LIN {X 0,Y 171.807,Z 301.135,A -85,B 0,C 180,E1 -23753.467,E2 -23753.467} C_VEL
LIN {X 0,Y 170.77,Z 299.112,A -85,B 0,C 180,E1 -23754.539,E2 -23754.539} C_VEL
LIN {X 0,Y 168.461,Z 295.33,A -85,B 0,C 180,E1 -23756.862,E2 -23756.862} C_VEL
LIN {X 0,Y 167.597,Z 293.95,A -85,B 0,C 180,E1 -23757.747,E2 -23757.747} C_VEL
LIN {X 0,Y 164.577,Z 289.423,A -85,B 0,C 180,E1 -23761.147,E2 -23761.147} C_VEL
LIN {X 0,Y 164.373,Z 288.892,A -85,B 0,C 180,E1 -23761.531,E2 -23761.531} C_VEL
LIN {X 0,Y 163.764,Z 286.973,A -85,B 0,C 180,E1 -23767.397,E2 -23767.397} C_VEL
LIN {X 0,Y 163.542,Z 286.029,A -85,B 0,C 180,E1 -23772.408,E2 -23772.408} C_VEL
LIN {X 0,Y 163.433,Z 285.855,A -85,B 0,C 180,E1 -23777.518,E2 -23777.518} C_VEL
LIN {X 0,Y 163.729,Z 286.439,A -85,B 0,C 180,E1 -23782.726,E2 -23782.726} C_VEL
LIN {X 0,Y 164.407,Z 287.979,A -85,B 0,C 180,E1 -23788.049,E2 -23788.049} C_VEL
LIN {X 0,Y 165.059,Z 289.593,A -85,B 0,C 180,E1 -23791.617,E2 -23791.617} C_VEL
LIN {X 0,Y 166.662,Z 293.516,A -85,B 0,C 180,E1 -23797.542,E2 -23797.542} C_VEL
LIN {X 0,Y 171.614,Z 300.55,A -85,B 0,C 180,E1 -23801.978,E2 -23801.978} C_VEL
LIN {X 0,Y 174.691,Z 306.548,A -85,B 0,C 180,E1 -23804.603,E2 -23804.603} C_VEL
LIN {X 0,Y 176.775,Z 311.643,A -85,B 0,C 180,E1 -23806.516,E2 -23806.516} C_VEL
LIN {X 0,Y 178.262,Z 321.519,A -85,B 0,C 180,E1 -23809.162,E2 -23809.162} C_VEL
LIN {X 0,Y 178.652,Z 330.917,A -85,B 0,C 180,E1 -23811.605,E2 -23811.605} C_VEL
LIN {X 0,Y 178.13,Z 336.639,A -85,B 0,C 180,E1 -23813.07,E2 -23813.07} C_VEL
LIN {X 0,Y 175.624,Z 345.707,A -85,B 0,C 180,E1 -23815.233,E2 -23815.233} C_VEL
LIN {X 0,Y 173.203,Z 353.233,A -85,B 0,C 180,E1 -23817.477,E2 -23817.477} C_VEL
LIN {X 0,Y 169.307,Z 361.018,A -85,B 0,C 180,E1 -23820.124,E2 -23820.124} C_VEL
LIN {X 0,Y 166.418,Z 366.182,A -85,B 0,C 180,E1 -23822.32,E2 -23822.32} C_VEL
LIN {X 0,Y 163.949,Z 370.527,A -85,B 0,C 180,E1 -23824.617,E2 -23824.617} C_VEL
LIN {X 0,Y 160.848,Z 375.707,A -85,B 0,C 180,E1 -23828.199,E2 -23828.199} C_VEL
LIN {X 0,Y 158.228,Z 379.6,A -85,B 0,C 180,E1 -23831.886,E2 -23831.886} C_VEL
LIN {X 0,Y 156.906,Z 381.458,A -85,B 0,C 180,E1 -23834.411,E2 -23834.411} C_VEL
LIN {X 0,Y 156.007,Z 382.844,A -85,B 0,C 180,E1 -23836.983,E2 -23836.983} C_VEL
LIN {X 0,Y 155.411,Z 383.78,A -85,B 0,C 180,E1 -23839.579,E2 -23839.579} C_VEL
LIN {X 0,Y 155.045,Z 384.215,A -85,B 0,C 180,E1 -23842.185,E2 -23842.185} C_VEL
LIN {X 0,Y 155.037,Z 383.994,A -85,B 0,C 180,E1 -23845.776,E2 -23845.776} C_VEL
LIN {X 0,Y 155.371,Z 382.438,A -85,B 0,C 180,E1 -23850,E2 -23850} C_VEL
LIN {X 0,Y 155.426,Z 380.832,A -85,B 0,C 180,E1 -23852.592,E2 -23852.592} C_VEL
LIN {X 0,Y 155.785,Z 377.198,A -85,B 0,C 180,E1 -23856.476,E2 -23856.476} C_VEL
LIN {X 0,Y 156.411,Z 374.594,A -85,B 0,C 180,E1 -23858.772,E2 -23858.772} C_VEL
LIN {X 0,Y 156.872,Z 377.363,A -85,B 0,C 180,E1 -23862.945,E2 -23862.945} C_VEL
LIN {X 0,Y 158.749,Z 379.707,A -85,B 0,C 180,E1 -23868.054,E2 -23868.054} C_VEL
LIN {X 0,Y 162.293,Z 380.986,A -85,B 0,C 180,E1 -23872.939,E2 -23872.939} C_VEL
LIN {X 0,Y 167.198,Z 381.193,A -85,B 0,C 180,E1 -23877.541,E2 -23877.541} C_VEL
LIN {X 0,Y 170.684,Z 380.806,A -85,B 0,C 180,E1 -23880.126,E2 -23880.126} C_VEL
LIN {X 0,Y 172.842,Z 380.336,A -85,B 0,C 180,E1 -23881.957,E2 -23881.957} C_VEL
LIN {X 0,Y 177.848,Z 378.2,A -85,B 0,C 180,E1 -23887.502,E2 -23887.502} C_VEL
LIN {X 0,Y 180.635,Z 377.227,A -85,B 0,C 180,E1 -23889.123,E2 -23889.123} C_VEL
LIN {X 0,Y 181.821,Z 376.834,A -85,B 0,C 180,E1 -23889.601,E2 -23889.601} C_VEL
LIN {X 0,Y 189.036,Z 374.503,A -85,B 0,C 180,E1 -23892.007,E2 -23892.007} C_VEL
LIN {X 0,Y 193.684,Z 372.683,A -85,B 0,C 180,E1 -23893.586,E2 -23893.586} C_VEL
LIN {X 0,Y 196.724,Z 371.102,A -85,B 0,C 180,E1 -23895.603,E2 -23895.603} C_VEL
LIN {X 0,Y 197.955,Z 370.173,A -85,B 0,C 180,E1 -23897.58,E2 -23897.58} C_VEL
LIN {X 0,Y 198.038,Z 370.015,A -85,B 0,C 180,E1 -23898.182,E2 -23898.182} C_VEL
LIN {X 0,Y 197.073,Z 370.011,A -85,B 0,C 180,E1 -23900.065,E2 -23900.065} C_VEL
LIN {X 0,Y 192.395,Z 371.253,A -85,B 0,C 180,E1 -23901.611,E2 -23901.611} C_VEL
LIN {X 0,Y 182.935,Z 373.108,A -85,B 0,C 180,E1 -23904.812,E2 -23904.812} C_VEL
LIN {X 0,Y 174.413,Z 373.822,A -85,B 0,C 180,E1 -23908.41,E2 -23908.41} C_VEL
LIN {X 0,Y 166.91,Z 373.402,A -85,B 0,C 180,E1 -23912.408,E2 -23912.408} C_VEL
LIN {X 0,Y 160.609,Z 371.833,A -85,B 0,C 180,E1 -23916.807,E2 -23916.807} C_VEL
LIN {X 0,Y 155.459,Z 369.106,A -85,B 0,C 180,E1 -23921.551,E2 -23921.551} C_VEL
LIN {X 0,Y 152.113,Z 365.227,A -85,B 0,C 180,E1 -23926.644,E2 -23926.644} C_VEL
LIN {X 0,Y 150.015,Z 360.025,A -85,B 0,C 180,E1 -23931.921,E2 -23931.921} C_VEL
LIN {X 0,Y 148.825,Z 353.277,A -85,B 0,C 180,E1 -23937.294,E2 -23937.294} C_VEL
LIN {X 0,Y 148.718,Z 345.944,A -85,B 0,C 180,E1 -23942.031,E2 -23942.031} C_VEL
LIN {X 0,Y 149.01,Z 337.459,A -85,B 0,C 180,E1 -23946.444,E2 -23946.444} C_VEL
LIN {X 0,Y 149.593,Z 328.841,A -85,B 0,C 180,E1 -23950.147,E2 -23950.147} C_VEL
LIN {X 0,Y 150.594,Z 317.422,A -85,B 0,C 180,E1 -23954.183,E2 -23954.183} C_VEL
LIN {X 0,Y 151.665,Z 306.976,A -85,B 0,C 180,E1 -23957.183,E2 -23957.183} C_VEL
LIN {X 0,Y 153,Z 294.302,A -85,B 0,C 180,E1 -23960.152,E2 -23960.152} C_VEL
LIN {X 0,Y 150.87,Z 281.95,A -85,B 0,C 180,E1 -23962.402,E2 -23962.402} C_VEL
LIN {X 0,Y 149.044,Z 269.969,A -85,B 0,C 180,E1 -23964.182,E2 -23964.182} C_VEL
LIN {X 0,Y 149.609,Z 269.848,A -85,B 0,C 180,E1 -23972.267,E2 -23972.267} C_VEL
LIN {X 0,Y 149.987,Z 269.803,A -85,B 0,C 180,E1 -23977.528,E2 -23977.528} C_VEL
LIN {X 0,Y 150.097,Z 269.785,A -85,B 0,C 180,E1 -23981.481,E2 -23981.481} C_VEL
LIN {X 0,Y 150.128,Z 269.785,A -85,B 0,C 180,E1 -23985.395,E2 -23985.395} C_VEL
LIN {X 0,Y 150.14,Z 269.784,A -85,B 0,C 180,E1 -23989.054,E2 -23989.054} C_VEL
LIN {X 0,Y 150.178,Z 269.777,A -85,B 0,C 180,E1 -23992.71,E2 -23992.71} C_VEL
LIN {X 0,Y 150.207,Z 269.774,A -85,B 0,C 180,E1 -23997.374,E2 -23997.374} C_VEL
LIN {X 0,Y 150.241,Z 269.771,A -85,B 0,C 180,E1 -24002.722,E2 -24002.722} C_VEL
LIN {X 0,Y 150.352,Z 269.756,A -85,B 0,C 180,E1 -24009.209,E2 -24009.209} C_VEL
LIN {X 0,Y 150.364,Z 269.748,A -85,B 0,C 180,E1 -24013.713,E2 -24013.713} C_VEL
LIN {X 0,Y 150.613,Z 269.726,A -85,B 0,C 180,E1 -24019.242,E2 -24019.242} C_VEL
LIN {X 0,Y 150.701,Z 269.791,A -85,B 0,C 180,E1 -24022.968,E2 -24022.968} C_VEL
LIN {X 0,Y 152.144,Z 275.605,A -85,B 0,C 180,E1 -24028.676,E2 -24028.676} C_VEL
LIN {X 0,Y 152.345,Z 278.494,A -85,B 0,C 180,E1 -24031.321,E2 -24031.321} C_VEL
LIN {X 0,Y 151.838,Z 283.129,A -85,B 0,C 180,E1 -24035.311,E2 -24035.311} C_VEL
LIN {X 0,Y 151.536,Z 285.299,A -85,B 0,C 180,E1 -24037.16,E2 -24037.16} C_VEL
LIN {X 0,Y 153.606,Z 296.207,A -85,B 0,C 180,E1 -24038.551,E2 -24038.551} C_VEL
LIN {X 0,Y 154.832,Z 304.081,A -85,B 0,C 180,E1 -24039.8,E2 -24039.8} C_VEL
LIN {X 0,Y 155.768,Z 312.475,A -85,B 0,C 180,E1 -24041.384,E2 -24041.384} C_VEL
LIN {X 0,Y 156.371,Z 319.655,A -85,B 0,C 180,E1 -24042.986,E2 -24042.986} C_VEL
LIN {X 0,Y 155.521,Z 325.645,A -85,B 0,C 180,E1 -24044.391,E2 -24044.391} C_VEL
LIN {X 0,Y 153.97,Z 333.329,A -85,B 0,C 180,E1 -24046.552,E2 -24046.552} C_VEL
LIN {X 0,Y 152.622,Z 339.884,A -85,B 0,C 180,E1 -24048.804,E2 -24048.804} C_VEL
LIN {X 0,Y 151.181,Z 346.539,A -85,B 0,C 180,E1 -24051.603,E2 -24051.603} C_VEL
LIN {X 0,Y 149.791,Z 352.955,A -85,B 0,C 180,E1 -24054.978,E2 -24054.978} C_VEL
LIN {X 0,Y 148.818,Z 357.754,A -85,B 0,C 180,E1 -24058.18,E2 -24058.18} C_VEL
LIN {X 0,Y 148.1,Z 361.611,A -85,B 0,C 180,E1 -24061.466,E2 -24061.466} C_VEL
LIN {X 0,Y 147.702,Z 365.391,A -85,B 0,C 180,E1 -24066.011,E2 -24066.011} C_VEL
LIN {X 0,Y 147.758,Z 366.729,A -85,B 0,C 180,E1 -24068.194,E2 -24068.194} C_VEL
LIN {X 0,Y 148.185,Z 368.093,A -85,B 0,C 180,E1 -24071.604,E2 -24071.604} C_VEL
LIN {X 0,Y 149.05,Z 368.678,A -85,B 0,C 180,E1 -24075.014,E2 -24075.014} C_VEL
LIN {X 0,Y 150.744,Z 368.281,A -85,B 0,C 180,E1 -24079.253,E2 -24079.253} C_VEL
LIN {X 0,Y 153.066,Z 366.635,A -85,B 0,C 180,E1 -24083.352,E2 -24083.352} C_VEL
LIN {X 0,Y 154.299,Z 365.627,A -85,B 0,C 180,E1 -24085.071,E2 -24085.071} C_VEL
LIN {X 0,Y 156.967,Z 362.887,A -85,B 0,C 180,E1 -24088.288,E2 -24088.288} C_VEL
LIN {X 0,Y 160.032,Z 359.11,A -85,B 0,C 180,E1 -24091.441,E2 -24091.441} C_VEL
LIN {X 0,Y 163.779,Z 353.917,A -85,B 0,C 180,E1 -24094.588,E2 -24094.588} C_VEL
LIN {X 0,Y 167.587,Z 347.987,A -85,B 0,C 180,E1 -24097.309,E2 -24097.309} C_VEL
LIN {X 0,Y 170.971,Z 341.922,A -85,B 0,C 180,E1 -24099.504,E2 -24099.504} C_VEL
LIN {X 0,Y 172.124,Z 339.009,A -85,B 0,C 180,E1 -24100.552,E2 -24100.552} C_VEL
LIN {X 0,Y 173.216,Z 331.259,A -85,B 0,C 180,E1 -24103.5,E2 -24103.5} C_VEL
LIN {X 0,Y 173.37,Z 324.684,A -85,B 0,C 180,E1 -24105.923,E2 -24105.923} C_VEL
LIN {X 0,Y 172.775,Z 318.629,A -85,B 0,C 180,E1 -24108.265,E2 -24108.265} C_VEL
LIN {X 0,Y 170.637,Z 312.341,A -85,B 0,C 180,E1 -24111.296,E2 -24111.296} C_VEL
LIN {X 0,Y 167.582,Z 305.138,A -85,B 0,C 180,E1 -24115.188,E2 -24115.188} C_VEL
LIN {X 0,Y 165.383,Z 301.117,A -85,B 0,C 180,E1 -24117.793,E2 -24117.793} C_VEL
LIN {X 0,Y 161.882,Z 295.216,A -85,B 0,C 180,E1 -24122.488,E2 -24122.488} C_VEL
LIN {X 0,Y 158.701,Z 291.959,A -85,B 0,C 180,E1 -24127.474,E2 -24127.474} C_VEL
LIN {X 0,Y 157.556,Z 290.073,A -85,B 0,C 180,E1 -24130.278,E2 -24130.278} C_VEL
LIN {X 0,Y 157.464,Z 289.678,A -85,B 0,C 180,E1 -24135.533,E2 -24135.533} C_VEL
LIN {X 0,Y 157.647,Z 290.116,A -85,B 0,C 180,E1 -24140.894,E2 -24140.894} C_VEL
LIN {X 0,Y 158.302,Z 291.389,A -85,B 0,C 180,E1 -24146.357,E2 -24146.357} C_VEL
LIN {X 0,Y 158.745,Z 292.495,A -85,B 0,C 180,E1 -24148.928,E2 -24148.928} C_VEL
LIN {X 0,Y 164.433,Z 300.122,A -85,B 0,C 180,E1 -24156.908,E2 -24156.908} C_VEL
LIN {X 0,Y 168.556,Z 306.487,A -85,B 0,C 180,E1 -24161.126,E2 -24161.126} C_VEL
LIN {X 0,Y 170.828,Z 311.443,A -85,B 0,C 180,E1 -24163.478,E2 -24163.478} C_VEL
LIN {X 0,Y 172.505,Z 316.408,A -85,B 0,C 180,E1 -24165.478,E2 -24165.478} C_VEL
LIN {X 0,Y 173.332,Z 325.826,A -85,B 0,C 180,E1 -24168.2,E2 -24168.2} C_VEL
LIN {X 0,Y 173.204,Z 333.712,A -85,B 0,C 180,E1 -24170.439,E2 -24170.439} C_VEL
LIN {X 0,Y 172.921,Z 337.214,A -85,B 0,C 180,E1 -24171.413,E2 -24171.413} C_VEL
LIN {X 0,Y 169.917,Z 346.903,A -85,B 0,C 180,E1 -24173.886,E2 -24173.886} C_VEL
LIN {X 0,Y 167.304,Z 354.116,A -85,B 0,C 180,E1 -24176.179,E2 -24176.179} C_VEL
LIN {X 0,Y 164.023,Z 360.283,A -85,B 0,C 180,E1 -24178.34,E2 -24178.34} C_VEL
LIN {X 0,Y 160.181,Z 366.633,A -85,B 0,C 180,E1 -24181.143,E2 -24181.143} C_VEL
LIN {X 0,Y 157.566,Z 370.826,A -85,B 0,C 180,E1 -24183.511,E2 -24183.511} C_VEL
LIN {X 0,Y 154.271,Z 375.865,A -85,B 0,C 180,E1 -24187.218,E2 -24187.218} C_VEL
LIN {X 0,Y 151.491,Z 379.605,A -85,B 0,C 180,E1 -24191.05,E2 -24191.05} C_VEL
LIN {X 0,Y 150.042,Z 381.346,A -85,B 0,C 180,E1 -24193.678,E2 -24193.678} C_VEL
LIN {X 0,Y 149.06,Z 382.615,A -85,B 0,C 180,E1 -24196.365,E2 -24196.365} C_VEL
LIN {X 0,Y 148.388,Z 383.441,A -85,B 0,C 180,E1 -24199.08,E2 -24199.08} C_VEL
LIN {X 0,Y 147.991,Z 383.82,A -85,B 0,C 180,E1 -24201.81,E2 -24201.81} C_VEL
LIN {X 0,Y 147.977,Z 383.385,A -85,B 0,C 180,E1 -24205.844,E2 -24205.844} C_VEL
LIN {X 0,Y 148.306,Z 381.789,A -85,B 0,C 180,E1 -24210,E2 -24210} C_VEL
LIN {X 0,Y 148.407,Z 378.972,A -85,B 0,C 180,E1 -24214.074,E2 -24214.074} C_VEL
LIN {X 0,Y 149.086,Z 374.871,A -85,B 0,C 180,E1 -24218.131,E2 -24218.131} C_VEL
LIN {X 0,Y 149.621,Z 373.086,A -85,B 0,C 180,E1 -24219.634,E2 -24219.634} C_VEL
LIN {X 0,Y 150.119,Z 375.704,A -85,B 0,C 180,E1 -24223.538,E2 -24223.538} C_VEL
LIN {X 0,Y 152.121,Z 378.357,A -85,B 0,C 180,E1 -24228.869,E2 -24228.869} C_VEL
LIN {X 0,Y 155.822,Z 379.961,A -85,B 0,C 180,E1 -24233.95,E2 -24233.95} C_VEL
LIN {X 0,Y 160.959,Z 380.526,A -85,B 0,C 180,E1 -24238.705,E2 -24238.705} C_VEL
LIN {X 0,Y 167.382,Z 380.073,A -85,B 0,C 180,E1 -24243.083,E2 -24243.083} C_VEL
LIN {X 0,Y 175.194,Z 378.621,A -85,B 0,C 180,E1 -24246.995,E2 -24246.995} C_VEL
LIN {X 0,Y 181.821,Z 376.834,A -85,B 0,C 180,E1 -24249.601,E2 -24249.601} C_VEL
LIN {X 0,Y 193.185,Z 372.928,A -85,B 0,C 180,E1 -24253.315,E2 -24253.315} C_VEL
LIN {X 0,Y 194.417,Z 372.367,A -85,B 0,C 180,E1 -24253.96,E2 -24253.96} C_VEL
LIN {X 0,Y 194.868,Z 371.948,A -85,B 0,C 180,E1 -24254.912,E2 -24254.912} C_VEL
LIN {X 0,Y 194.1,Z 371.779,A -85,B 0,C 180,E1 -24256.298,E2 -24256.298} C_VEL
LIN {X 0,Y 191.77,Z 372.044,A -85,B 0,C 180,E1 -24257.97,E2 -24257.97} C_VEL
LIN {X 0,Y 188.64,Z 372.559,A -85,B 0,C 180,E1 -24259.544,E2 -24259.544} C_VEL
LIN {X 0,Y 186.99,Z 372.866,A -85,B 0,C 180,E1 -24260.287,E2 -24260.287} C_VEL
LIN {X 0,Y 177.233,Z 374.236,A -85,B 0,C 180,E1 -24263.501,E2 -24263.501} C_VEL
LIN {X 0,Y 168.427,Z 374.487,A -85,B 0,C 180,E1 -24267.149,E2 -24267.149} C_VEL
LIN {X 0,Y 160.661,Z 373.62,A -85,B 0,C 180,E1 -24271.237,E2 -24271.237} C_VEL
LIN {X 0,Y 154.111,Z 371.633,A -85,B 0,C 180,E1 -24275.768,E2 -24275.768} C_VEL
LIN {X 0,Y 148.775,Z 368.506,A -85,B 0,C 180,E1 -24280.69,E2 -24280.69} C_VEL
LIN {X 0,Y 145.282,Z 364.241,A -85,B 0,C 180,E1 -24286.003,E2 -24286.003} C_VEL
LIN {X 0,Y 143.116,Z 358.694,A -85,B 0,C 180,E1 -24291.529,E2 -24291.529} C_VEL
LIN {X 0,Y 141.911,Z 351.525,A -85,B 0,C 180,E1 -24297.162,E2 -24297.162} C_VEL
LIN {X 0,Y 141.817,Z 344.989,A -85,B 0,C 180,E1 -24301.42,E2 -24301.42} C_VEL
LIN {X 0,Y 142.044,Z 337.093,A -85,B 0,C 180,E1 -24305.679,E2 -24305.679} C_VEL
LIN {X 0,Y 142.578,Z 328.22,A -85,B 0,C 180,E1 -24309.647,E2 -24309.647} C_VEL
LIN {X 0,Y 143.562,Z 316.905,A -85,B 0,C 180,E1 -24313.807,E2 -24313.807} C_VEL
LIN {X 0,Y 144.742,Z 305.089,A -85,B 0,C 180,E1 -24317.302,E2 -24317.302} C_VEL
LIN {X 0,Y 145.846,Z 293.735,A -85,B 0,C 180,E1 -24320.046,E2 -24320.046} C_VEL
LIN {X 0,Y 143.451,Z 280.113,A -85,B 0,C 180,E1 -24322.57,E2 -24322.57} C_VEL
LIN {X 0,Y 142.01,Z 270.797,A -85,B 0,C 180,E1 -24324.001,E2 -24324.001} C_VEL
LIN {X 0,Y 142.251,Z 270.764,A -85,B 0,C 180,E1 -24329.608,E2 -24329.608} C_VEL
LIN {X 0,Y 142.62,Z 270.717,A -85,B 0,C 180,E1 -24333.098,E2 -24333.098} C_VEL
LIN {X 0,Y 142.923,Z 270.682,A -85,B 0,C 180,E1 -24338.114,E2 -24338.114} C_VEL
LIN {X 0,Y 143.025,Z 270.672,A -85,B 0,C 180,E1 -24343.468,E2 -24343.468} C_VEL
LIN {X 0,Y 143.04,Z 270.664,A -85,B 0,C 180,E1 -24347.477,E2 -24347.477} C_VEL
LIN {X 0,Y 143.074,Z 270.664,A -85,B 0,C 180,E1 -24351.809,E2 -24351.809} C_VEL
LIN {X 0,Y 143.175,Z 270.65,A -85,B 0,C 180,E1 -24357.319,E2 -24357.319} C_VEL
LIN {X 0,Y 143.185,Z 270.65,A -85,B 0,C 180,E1 -24362.069,E2 -24362.069} C_VEL
LIN {X 0,Y 143.278,Z 270.638,A -85,B 0,C 180,E1 -24368.747,E2 -24368.747} C_VEL
LIN {X 0,Y 143.304,Z 270.624,A -85,B 0,C 180,E1 -24372.886,E2 -24372.886} C_VEL
LIN {X 0,Y 143.539,Z 270.604,A -85,B 0,C 180,E1 -24378.705,E2 -24378.705} C_VEL
LIN {X 0,Y 143.679,Z 270.713,A -85,B 0,C 180,E1 -24381.915,E2 -24381.915} C_VEL
LIN {X 0,Y 145.241,Z 277.269,A -85,B 0,C 180,E1 -24388.613,E2 -24388.613} C_VEL
LIN {X 0,Y 145.388,Z 280.234,A -85,B 0,C 180,E1 -24391.385,E2 -24391.385} C_VEL
LIN {X 0,Y 144.683,Z 285.645,A -85,B 0,C 180,E1 -24396.187,E2 -24396.187} C_VEL
LIN {X 0,Y 146.749,Z 296.639,A -85,B 0,C 180,E1 -24397.654,E2 -24397.654} C_VEL
LIN {X 0,Y 148.158,Z 305.851,A -85,B 0,C 180,E1 -24399.212,E2 -24399.212} C_VEL
LIN {X 0,Y 149.139,Z 315.612,A -85,B 0,C 180,E1 -24401.208,E2 -24401.208} C_VEL
LIN {X 0,Y 149.475,Z 321.134,A -85,B 0,C 180,E1 -24402.559,E2 -24402.559} C_VEL
LIN {X 0,Y 147.825,Z 329.804,A -85,B 0,C 180,E1 -24404.805,E2 -24404.805} C_VEL
LIN {X 0,Y 146.118,Z 338.047,A -85,B 0,C 180,E1 -24407.494,E2 -24407.494} C_VEL
LIN {X 0,Y 144.469,Z 345.364,A -85,B 0,C 180,E1 -24410.546,E2 -24410.546} C_VEL
LIN {X 0,Y 143.039,Z 351.765,A -85,B 0,C 180,E1 -24413.913,E2 -24413.913} C_VEL
LIN {X 0,Y 142.009,Z 356.514,A -85,B 0,C 180,E1 -24417.022,E2 -24417.022} C_VEL
LIN {X 0,Y 141.082,Z 361.178,A -85,B 0,C 180,E1 -24420.914,E2 -24420.914} C_VEL
LIN {X 0,Y 140.636,Z 364.881,A -85,B 0,C 180,E1 -24425.078,E2 -24425.078} C_VEL
LIN {X 0,Y 140.899,Z 367.803,A -85,B 0,C 180,E1 -24430.423,E2 -24430.423} C_VEL
LIN {X 0,Y 141.62,Z 368.809,A -85,B 0,C 180,E1 -24434.008,E2 -24434.008} C_VEL
LIN {X 0,Y 142.813,Z 369.031,A -85,B 0,C 180,E1 -24437.575,E2 -24437.575} C_VEL
LIN {X 0,Y 144.494,Z 368.463,A -85,B 0,C 180,E1 -24441.098,E2 -24441.098} C_VEL
LIN {X 0,Y 147.951,Z 366.08,A -85,B 0,C 180,E1 -24446.353,E2 -24446.353} C_VEL
LIN {X 0,Y 151.119,Z 362.993,A -85,B 0,C 180,E1 -24450.041,E2 -24450.041} C_VEL
LIN {X 0,Y 154.779,Z 358.723,A -85,B 0,C 180,E1 -24453.53,E2 -24453.53} C_VEL
LIN {X 0,Y 158.579,Z 353.787,A -85,B 0,C 180,E1 -24456.492,E2 -24456.492} C_VEL
LIN {X 0,Y 162.895,Z 347.427,A -85,B 0,C 180,E1 -24459.387,E2 -24459.387} C_VEL
LIN {X 0,Y 165.436,Z 343.103,A -85,B 0,C 180,E1 -24460.957,E2 -24460.957} C_VEL
LIN {X 0,Y 166.599,Z 339.938,A -85,B 0,C 180,E1 -24462.25,E2 -24462.25} C_VEL
LIN {X 0,Y 167.825,Z 332.05,A -85,B 0,C 180,E1 -24465.447,E2 -24465.447} C_VEL
LIN {X 0,Y 168.122,Z 325.849,A -85,B 0,C 180,E1 -24467.935,E2 -24467.935} C_VEL
LIN {X 0,Y 167.604,Z 321.749,A -85,B 0,C 180,E1 -24469.772,E2 -24469.772} C_VEL
LIN {X 0,Y 165.583,Z 315.244,A -85,B 0,C 180,E1 -24473.297,E2 -24473.297} C_VEL
LIN {X 0,Y 163.637,Z 310.341,A -85,B 0,C 180,E1 -24476.306,E2 -24476.306} C_VEL
LIN {X 0,Y 161.264,Z 305.387,A -85,B 0,C 180,E1 -24480,E2 -24480} C_VEL
LIN {X 0,Y 159.406,Z 301.654,A -85,B 0,C 180,E1 -24483.159,E2 -24483.159} C_VEL
LIN {X 0,Y 156.829,Z 298.625,A -85,B 0,C 180,E1 -24488.043,E2 -24488.043} C_VEL
LIN {X 0,Y 155.867,Z 296.907,A -85,B 0,C 180,E1 -24490.785,E2 -24490.785} C_VEL
LIN {X 0,Y 154.56,Z 296.202,A -85,B 0,C 180,E1 -24497.275,E2 -24497.275} C_VEL
LIN {X 0,Y 155.145,Z 297.123,A -85,B 0,C 180,E1 -24503.351,E2 -24503.351} C_VEL
LIN {X 0,Y 156.989,Z 299.239,A -85,B 0,C 180,E1 -24508.416,E2 -24508.416} C_VEL
LIN {X 0,Y 161.888,Z 306.537,A -85,B 0,C 180,E1 -24516.263,E2 -24516.263} C_VEL
LIN {X 0,Y 164.993,Z 311.624,A -85,B 0,C 180,E1 -24519.939,E2 -24519.939} C_VEL
LIN {X 0,Y 167.257,Z 317.894,A -85,B 0,C 180,E1 -24523.064,E2 -24523.064} C_VEL
LIN {X 0,Y 168.166,Z 321.202,A -85,B 0,C 180,E1 -24524.43,E2 -24524.43} C_VEL
LIN {X 0,Y 168.25,Z 331.7,A -85,B 0,C 180,E1 -24527.716,E2 -24527.716} C_VEL
LIN {X 0,Y 167.536,Z 338.916,A -85,B 0,C 180,E1 -24529.927,E2 -24529.927} C_VEL
LIN {X 0,Y 165.062,Z 346.196,A -85,B 0,C 180,E1 -24531.875,E2 -24531.875} C_VEL
LIN {X 0,Y 162.266,Z 353.413,A -85,B 0,C 180,E1 -24534.218,E2 -24534.218} C_VEL
LIN {X 0,Y 158.925,Z 359.605,A -85,B 0,C 180,E1 -24536.442,E2 -24536.442} C_VEL
LIN {X 0,Y 154.792,Z 365.997,A -85,B 0,C 180,E1 -24539.284,E2 -24539.284} C_VEL
LIN {X 0,Y 152.49,Z 369.354,A -85,B 0,C 180,E1 -24541.125,E2 -24541.125} C_VEL
LIN {X 0,Y 148.786,Z 374.513,A -85,B 0,C 180,E1 -24544.842,E2 -24544.842} C_VEL
LIN {X 0,Y 145.672,Z 378.469,A -85,B 0,C 180,E1 -24548.787,E2 -24548.787} C_VEL
LIN {X 0,Y 143.209,Z 381.249,A -85,B 0,C 180,E1 -24552.876,E2 -24552.876} C_VEL
LIN {X 0,Y 142.141,Z 382.398,A -85,B 0,C 180,E1 -24555.687,E2 -24555.687} C_VEL
LIN {X 0,Y 141.39,Z 383.105,A -85,B 0,C 180,E1 -24558.532,E2 -24558.532} C_VEL
LIN {X 0,Y 140.959,Z 383.378,A -85,B 0,C 180,E1 -24561.398,E2 -24561.398} C_VEL
LIN {X 0,Y 140.92,Z 382.758,A -85,B 0,C 180,E1 -24565.905,E2 -24565.905} C_VEL
LIN {X 0,Y 141.242,Z 381.13,A -85,B 0,C 180,E1 -24570,E2 -24570} C_VEL
LIN {X 0,Y 141.37,Z 378.201,A -85,B 0,C 180,E1 -24574.277,E2 -24574.277} C_VEL
LIN {X 0,Y 142.133,Z 373.909,A -85,B 0,C 180,E1 -24578.531,E2 -24578.531} C_VEL
LIN {X 0,Y 142.931,Z 371.413,A -85,B 0,C 180,E1 -24580.537,E2 -24580.537} C_VEL
LIN {X 0,Y 144.27,Z 375.536,A -85,B 0,C 180,E1 -24586.995,E2 -24586.995} C_VEL
LIN {X 0,Y 147.273,Z 377.973,A -85,B 0,C 180,E1 -24592.444,E2 -24592.444} C_VEL
LIN {X 0,Y 151.905,Z 379.387,A -85,B 0,C 180,E1 -24597.559,E2 -24597.559} C_VEL
LIN {X 0,Y 157.935,Z 379.801,A -85,B 0,C 180,E1 -24602.276,E2 -24602.276} C_VEL
LIN {X 0,Y 165.338,Z 379.252,A -85,B 0,C 180,E1 -24606.52,E2 -24606.52} C_VEL
LIN {X 0,Y 174.109,Z 377.723,A -85,B 0,C 180,E1 -24610.23,E2 -24610.23} C_VEL
LIN {X 0,Y 183.85,Z 375.192,A -85,B 0,C 180,E1 -24613.479,E2 -24613.479} C_VEL
LIN {X 0,Y 188.392,Z 373.65,A -85,B 0,C 180,E1 -24615.138,E2 -24615.138} C_VEL
LIN {X 0,Y 190.893,Z 372.403,A -85,B 0,C 180,E1 -24617.42,E2 -24617.42} C_VEL
LIN {X 0,Y 191.006,Z 372.128,A -85,B 0,C 180,E1 -24618.524,E2 -24618.524} C_VEL
LIN {X 0,Y 188.64,Z 372.559,A -85,B 0,C 180,E1 -24619.544,E2 -24619.544} C_VEL
LIN {X 0,Y 186.325,Z 373.029,A -85,B 0,C 180,E1 -24620.237,E2 -24620.237} C_VEL
LIN {X 0,Y 182.184,Z 373.821,A -85,B 0,C 180,E1 -24620.871,E2 -24620.871} C_VEL
LIN {X 0,Y 173.219,Z 375.04,A -85,B 0,C 180,E1 -24621.899,E2 -24621.899} C_VEL
LIN {X 0,Y 169.993,Z 375.2,A -85,B 0,C 180,E1 -24622.709,E2 -24622.709} C_VEL
LIN {X 0,Y 162.529,Z 374.98,A -85,B 0,C 180,E1 -24625.796,E2 -24625.796} C_VEL
LIN {X 0,Y 154.472,Z 373.673,A -85,B 0,C 180,E1 -24629.969,E2 -24629.969} C_VEL
LIN {X 0,Y 147.683,Z 371.272,A -85,B 0,C 180,E1 -24634.641,E2 -24634.641} C_VEL
LIN {X 0,Y 142.148,Z 367.74,A -85,B 0,C 180,E1 -24639.752,E2 -24639.752} C_VEL
LIN {X 0,Y 138.512,Z 363.094,A -85,B 0,C 180,E1 -24645.304,E2 -24645.304} C_VEL
LIN {X 0,Y 136.241,Z 357.148,A -85,B 0,C 180,E1 -24651.098,E2 -24651.098} C_VEL
LIN {X 0,Y 135.054,Z 349.606,A -85,B 0,C 180,E1 -24657.017,E2 -24657.017} C_VEL
LIN {X 0,Y 134.959,Z 342.701,A -85,B 0,C 180,E1 -24661.492,E2 -24661.492} C_VEL
LIN {X 0,Y 135.202,Z 334.358,A -85,B 0,C 180,E1 -24665.968,E2 -24665.968} C_VEL
LIN {X 0,Y 135.773,Z 324.969,A -85,B 0,C 180,E1 -24670.135,E2 -24670.135} C_VEL
LIN {X 0,Y 136.749,Z 314.063,A -85,B 0,C 180,E1 -24674.13,E2 -24674.13} C_VEL
LIN {X 0,Y 137.987,Z 301.65,A -85,B 0,C 180,E1 -24677.794,E2 -24677.794} C_VEL
LIN {X 0,Y 138.706,Z 293.442,A -85,B 0,C 180,E1 -24679.807,E2 -24679.807} C_VEL
LIN {X 0,Y 136.238,Z 279.723,A -85,B 0,C 180,E1 -24682.454,E2 -24682.454} C_VEL
LIN {X 0,Y 134.981,Z 271.673,A -85,B 0,C 180,E1 -24683.803,E2 -24683.803} C_VEL
LIN {X 0,Y 135.339,Z 271.627,A -85,B 0,C 180,E1 -24691.285,E2 -24691.285} C_VEL
LIN {X 0,Y 135.633,Z 271.583,A -85,B 0,C 180,E1 -24694.749,E2 -24694.749} C_VEL
LIN {X 0,Y 135.922,Z 271.554,A -85,B 0,C 180,E1 -24699.14,E2 -24699.14} C_VEL
LIN {X 0,Y 135.971,Z 271.55,A -85,B 0,C 180,E1 -24703.644,E2 -24703.644} C_VEL
LIN {X 0,Y 135.984,Z 271.543,A -85,B 0,C 180,E1 -24707.787,E2 -24707.787} C_VEL
LIN {X 0,Y 136.023,Z 271.542,A -85,B 0,C 180,E1 -24711.682,E2 -24711.682} C_VEL
LIN {X 0,Y 136.053,Z 271.539,A -85,B 0,C 180,E1 -24715.742,E2 -24715.742} C_VEL
LIN {X 0,Y 136.142,Z 271.527,A -85,B 0,C 180,E1 -24722.315,E2 -24722.315} C_VEL
LIN {X 0,Y 136.244,Z 271.514,A -85,B 0,C 180,E1 -24728.832,E2 -24728.832} C_VEL
LIN {X 0,Y 136.271,Z 271.511,A -85,B 0,C 180,E1 -24735.056,E2 -24735.056} C_VEL
LIN {X 0,Y 136.536,Z 271.541,A -85,B 0,C 180,E1 -24740.658,E2 -24740.658} C_VEL
LIN {X 0,Y 137.529,Z 276.19,A -85,B 0,C 180,E1 -24745.603,E2 -24745.603} C_VEL
LIN {X 0,Y 138.354,Z 278.95,A -85,B 0,C 180,E1 -24748.544,E2 -24748.544} C_VEL
LIN {X 0,Y 138.416,Z 281.946,A -85,B 0,C 180,E1 -24751.454,E2 -24751.454} C_VEL
LIN {X 0,Y 137.878,Z 286.1,A -85,B 0,C 180,E1 -24755.117,E2 -24755.117} C_VEL
LIN {X 0,Y 139.847,Z 296.491,A -85,B 0,C 180,E1 -24756.583,E2 -24756.583} C_VEL
LIN {X 0,Y 141.248,Z 305.754,A -85,B 0,C 180,E1 -24758.224,E2 -24758.224} C_VEL
LIN {X 0,Y 142.218,Z 315.545,A -85,B 0,C 180,E1 -24760.319,E2 -24760.319} C_VEL
LIN {X 0,Y 142.498,Z 322.535,A -85,B 0,C 180,E1 -24762.099,E2 -24762.099} C_VEL
LIN {X 0,Y 140.485,Z 332.225,A -85,B 0,C 180,E1 -24764.813,E2 -24764.813} C_VEL
LIN {X 0,Y 138.721,Z 340.095,A -85,B 0,C 180,E1 -24767.696,E2 -24767.696} C_VEL
LIN {X 0,Y 137.031,Z 347.358,A -85,B 0,C 180,E1 -24771.039,E2 -24771.039} C_VEL
LIN {X 0,Y 135.443,Z 354.503,A -85,B 0,C 180,E1 -24775.232,E2 -24775.232} C_VEL
LIN {X 0,Y 134.197,Z 360.266,A -85,B 0,C 180,E1 -24779.836,E2 -24779.836} C_VEL
LIN {X 0,Y 133.605,Z 364.068,A -85,B 0,C 180,E1 -24783.952,E2 -24783.952} C_VEL
LIN {X 0,Y 133.647,Z 367.385,A -85,B 0,C 180,E1 -24789.126,E2 -24789.126} C_VEL
LIN {X 0,Y 134.234,Z 368.809,A -85,B 0,C 180,E1 -24792.893,E2 -24792.893} C_VEL
LIN {X 0,Y 135.686,Z 369.512,A -85,B 0,C 180,E1 -24797.673,E2 -24797.673} C_VEL
LIN {X 0,Y 137.918,Z 368.89,A -85,B 0,C 180,E1 -24802.302,E2 -24802.302} C_VEL
LIN {X 0,Y 140.828,Z 367.101,A -85,B 0,C 180,E1 -24806.704,E2 -24806.704} C_VEL
LIN {X 0,Y 144.589,Z 363.995,A -85,B 0,C 180,E1 -24811.035,E2 -24811.035} C_VEL
LIN {X 0,Y 148.656,Z 359.731,A -85,B 0,C 180,E1 -24814.818,E2 -24814.818} C_VEL
LIN {X 0,Y 152.157,Z 355.625,A -85,B 0,C 180,E1 -24817.485,E2 -24817.485} C_VEL
LIN {X 0,Y 156.602,Z 349.576,A -85,B 0,C 180,E1 -24820.465,E2 -24820.465} C_VEL
LIN {X 0,Y 159.959,Z 344.386,A -85,B 0,C 180,E1 -24822.487,E2 -24822.487} C_VEL
LIN {X 0,Y 161.247,Z 340.668,A -85,B 0,C 180,E1 -24824.168,E2 -24824.168} C_VEL
LIN {X 0,Y 162.657,Z 332.986,A -85,B 0,C 180,E1 -24827.523,E2 -24827.523} C_VEL
LIN {X 0,Y 162.89,Z 327.372,A -85,B 0,C 180,E1 -24830.062,E2 -24830.062} C_VEL
LIN {X 0,Y 161.718,Z 322.019,A -85,B 0,C 180,E1 -24833.136,E2 -24833.136} C_VEL
LIN {X 0,Y 160.241,Z 317.157,A -85,B 0,C 180,E1 -24836.228,E2 -24836.228} C_VEL
LIN {X 0,Y 158.389,Z 312.094,A -85,B 0,C 180,E1 -24840,E2 -24840} C_VEL
LIN {X 0,Y 157.159,Z 309.236,A -85,B 0,C 180,E1 -24842.563,E2 -24842.563} C_VEL
LIN {X 0,Y 153.859,Z 303.69,A -85,B 0,C 180,E1 -24851.027,E2 -24851.027} C_VEL
LIN {X 0,Y 152.874,Z 303.087,A -85,B 0,C 180,E1 -24856.012,E2 -24856.012} C_VEL
LIN {X 0,Y 153.046,Z 303.614,A -85,B 0,C 180,E1 -24861.553,E2 -24861.553} C_VEL
LIN {X 0,Y 154.678,Z 305.543,A -85,B 0,C 180,E1 -24867.39,E2 -24867.39} C_VEL
LIN {X 0,Y 158.72,Z 312.183,A -85,B 0,C 180,E1 -24875.144,E2 -24875.144} C_VEL
LIN {X 0,Y 161.377,Z 317.381,A -85,B 0,C 180,E1 -24879.157,E2 -24879.157} C_VEL
LIN {X 0,Y 162.985,Z 322.567,A -85,B 0,C 180,E1 -24881.943,E2 -24881.943} C_VEL
LIN {X 0,Y 163.481,Z 324.906,A -85,B 0,C 180,E1 -24883.045,E2 -24883.045} C_VEL
LIN {X 0,Y 163.327,Z 332.167,A -85,B 0,C 180,E1 -24885.534,E2 -24885.534} C_VEL
LIN {X 0,Y 162.52,Z 338.956,A -85,B 0,C 180,E1 -24887.801,E2 -24887.801} C_VEL
LIN {X 0,Y 161.811,Z 342.119,A -85,B 0,C 180,E1 -24888.816,E2 -24888.816} C_VEL
LIN {X 0,Y 158.11,Z 351.192,A -85,B 0,C 180,E1 -24891.516,E2 -24891.516} C_VEL
LIN {X 0,Y 154.89,Z 357.586,A -85,B 0,C 180,E1 -24893.853,E2 -24893.853} C_VEL
LIN {X 0,Y 150.457,Z 364.223,A -85,B 0,C 180,E1 -24896.712,E2 -24896.712} C_VEL
LIN {X 0,Y 146.953,Z 368.913,A -85,B 0,C 180,E1 -24899.26,E2 -24899.26} C_VEL
LIN {X 0,Y 143.665,Z 373.197,A -85,B 0,C 180,E1 -24902.307,E2 -24902.307} C_VEL
LIN {X 0,Y 140.124,Z 377.35,A -85,B 0,C 180,E1 -24906.344,E2 -24906.344} C_VEL
LIN {X 0,Y 138.083,Z 379.472,A -85,B 0,C 180,E1 -24909.129,E2 -24909.129} C_VEL
LIN {X 0,Y 136.406,Z 381.108,A -85,B 0,C 180,E1 -24911.993,E2 -24911.993} C_VEL
LIN {X 0,Y 135.231,Z 382.184,A -85,B 0,C 180,E1 -24914.939,E2 -24914.939} C_VEL
LIN {X 0,Y 134.419,Z 382.773,A -85,B 0,C 180,E1 -24917.929,E2 -24917.929} C_VEL
LIN {X 0,Y 133.924,Z 382.927,A -85,B 0,C 180,E1 -24920.943,E2 -24920.943} C_VEL
LIN {X 0,Y 133.771,Z 382.645,A -85,B 0,C 180,E1 -24923.969,E2 -24923.969} C_VEL
LIN {X 0,Y 133.973,Z 381.85,A -85,B 0,C 180,E1 -24926.993,E2 -24926.993} C_VEL
LIN {X 0,Y 134.179,Z 380.463,A -85,B 0,C 180,E1 -24930,E2 -24930} C_VEL
LIN {X 0,Y 134.336,Z 377.418,A -85,B 0,C 180,E1 -24934.501,E2 -24934.501} C_VEL
LIN {X 0,Y 135.186,Z 372.891,A -85,B 0,C 180,E1 -24938.973,E2 -24938.973} C_VEL
LIN {X 0,Y 136.32,Z 369.723,A -85,B 0,C 180,E1 -24941.609,E2 -24941.609} C_VEL
LIN {X 0,Y 137.685,Z 373.762,A -85,B 0,C 180,E1 -24947.835,E2 -24947.835} C_VEL
LIN {X 0,Y 140.857,Z 376.51,A -85,B 0,C 180,E1 -24953.526,E2 -24953.526} C_VEL
LIN {X 0,Y 145.735,Z 378.263,A -85,B 0,C 180,E1 -24958.833,E2 -24958.833} C_VEL
LIN {X 0,Y 152.008,Z 379.029,A -85,B 0,C 180,E1 -24963.699,E2 -24963.699} C_VEL
LIN {X 0,Y 159.698,Z 378.87,A -85,B 0,C 180,E1 -24968.034,E2 -24968.034} C_VEL
LIN {X 0,Y 168.751,Z 377.774,A -85,B 0,C 180,E1 -24971.787,E2 -24971.787} C_VEL
LIN {X 0,Y 178.787,Z 375.704,A -85,B 0,C 180,E1 -24975.038,E2 -24975.038} C_VEL
LIN {X 0,Y 182.925,Z 374.458,A -85,B 0,C 180,E1 -24976.886,E2 -24976.886} C_VEL
LIN {X 0,Y 183.311,Z 374.087,A -85,B 0,C 180,E1 -24978.172,E2 -24978.172} C_VEL
LIN {X 0,Y 181.663,Z 374.296,A -85,B 0,C 180,E1 -24978.877,E2 -24978.877} C_VEL
LIN {X 0,Y 171.624,Z 375.189,A -85,B 0,C 180,E1 -24982.103,E2 -24982.103} C_VEL
LIN {X 0,Y 169.993,Z 375.2,A -85,B 0,C 180,E1 -24982.709,E2 -24982.709} C_VEL
LIN {X 0,Y 165.649,Z 375.242,A -85,B 0,C 180,E1 -24984.078,E2 -24984.078} C_VEL
LIN {X 0,Y 157.493,Z 374.879,A -85,B 0,C 180,E1 -24986.074,E2 -24986.074} C_VEL
LIN {X 0,Y 149.698,Z 373.754,A -85,B 0,C 180,E1 -24988.303,E2 -24988.303} C_VEL
LIN {X 0,Y 146.013,Z 372.748,A -85,B 0,C 180,E1 -24990.041,E2 -24990.041} C_VEL
LIN {X 0,Y 138.294,Z 368.917,A -85,B 0,C 180,E1 -24996.012,E2 -24996.012} C_VEL
LIN {X 0,Y 133.471,Z 364.437,A -85,B 0,C 180,E1 -25001.583,E2 -25001.583} C_VEL
LIN {X 0,Y 130.447,Z 358.778,A -85,B 0,C 180,E1 -25007.555,E2 -25007.555} C_VEL
LIN {X 0,Y 128.956,Z 353.602,A -85,B 0,C 180,E1 -25012.17,E2 -25012.17} C_VEL
LIN {X 0,Y 128.166,Z 345.164,A -85,B 0,C 180,E1 -25018.429,E2 -25018.429} C_VEL
LIN {X 0,Y 128.198,Z 337.421,A -85,B 0,C 180,E1 -25023.143,E2 -25023.143} C_VEL
LIN {X 0,Y 128.583,Z 328.415,A -85,B 0,C 180,E1 -25027.681,E2 -25027.681} C_VEL
LIN {X 0,Y 129.236,Z 318.524,A -85,B 0,C 180,E1 -25031.797,E2 -25031.797} C_VEL
LIN {X 0,Y 130.363,Z 307.33,A -85,B 0,C 180,E1 -25035.638,E2 -25035.638} C_VEL
LIN {X 0,Y 131.629,Z 294.899,A -85,B 0,C 180,E1 -25039.089,E2 -25039.089} C_VEL
LIN {X 0,Y 130.974,Z 289.886,A -85,B 0,C 180,E1 -25040.209,E2 -25040.209} C_VEL
LIN {X 0,Y 128.435,Z 275.373,A -85,B 0,C 180,E1 -25042.948,E2 -25042.948} C_VEL
LIN {X 0,Y 127.991,Z 272.543,A -85,B 0,C 180,E1 -25043.46,E2 -25043.46} C_VEL
LIN {X 0,Y 128.116,Z 272.524,A -85,B 0,C 180,E1 -25049.585,E2 -25049.585} C_VEL
LIN {X 0,Y 128.588,Z 272.461,A -85,B 0,C 180,E1 -25054.931,E2 -25054.931} C_VEL
LIN {X 0,Y 128.852,Z 272.43,A -85,B 0,C 180,E1 -25060.884,E2 -25060.884} C_VEL
LIN {X 0,Y 128.912,Z 272.429,A -85,B 0,C 180,E1 -25065.133,E2 -25065.133} C_VEL
LIN {X 0,Y 128.936,Z 272.427,A -85,B 0,C 180,E1 -25069.74,E2 -25069.74} C_VEL
LIN {X 0,Y 128.957,Z 272.422,A -85,B 0,C 180,E1 -25074.834,E2 -25074.834} C_VEL
LIN {X 0,Y 129.019,Z 272.415,A -85,B 0,C 180,E1 -25080.642,E2 -25080.642} C_VEL
LIN {X 0,Y 129.11,Z 272.398,A -85,B 0,C 180,E1 -25087.601,E2 -25087.601} C_VEL
LIN {X 0,Y 129.155,Z 272.391,A -85,B 0,C 180,E1 -25090.943,E2 -25090.943} C_VEL
LIN {X 0,Y 129.369,Z 272.365,A -85,B 0,C 180,E1 -25097.923,E2 -25097.923} C_VEL
LIN {X 0,Y 129.47,Z 272.48,A -85,B 0,C 180,E1 -25099.337,E2 -25099.337} C_VEL
LIN {X 0,Y 130.352,Z 276.413,A -85,B 0,C 180,E1 -25103.809,E2 -25103.809} C_VEL
LIN {X 0,Y 131.474,Z 280.65,A -85,B 0,C 180,E1 -25108.468,E2 -25108.468} C_VEL
LIN {X 0,Y 131.448,Z 283.722,A -85,B 0,C 180,E1 -25111.531,E2 -25111.531} C_VEL
LIN {X 0,Y 131.048,Z 286.28,A -85,B 0,C 180,E1 -25113.94,E2 -25113.94} C_VEL
LIN {X 0,Y 133.107,Z 297.252,A -85,B 0,C 180,E1 -25115.586,E2 -25115.586} C_VEL
LIN {X 0,Y 134.362,Z 305.578,A -85,B 0,C 180,E1 -25117.136,E2 -25117.136} C_VEL
LIN {X 0,Y 135.188,Z 313.935,A -85,B 0,C 180,E1 -25118.972,E2 -25118.972} C_VEL
LIN {X 0,Y 135.679,Z 322.445,A -85,B 0,C 180,E1 -25121.2,E2 -25121.2} C_VEL
LIN {X 0,Y 133.866,Z 331.047,A -85,B 0,C 180,E1 -25123.665,E2 -25123.665} C_VEL
LIN {X 0,Y 131.865,Z 339.896,A -85,B 0,C 180,E1 -25126.942,E2 -25126.942} C_VEL
LIN {X 0,Y 130.012,Z 347.462,A -85,B 0,C 180,E1 -25130.571,E2 -25130.571} C_VEL
LIN {X 0,Y 128.92,Z 352.081,A -85,B 0,C 180,E1 -25133.278,E2 -25133.278} C_VEL
LIN {X 0,Y 127.727,Z 357.32,A -85,B 0,C 180,E1 -25137.064,E2 -25137.064} C_VEL
LIN {X 0,Y 126.757,Z 362.284,A -85,B 0,C 180,E1 -25141.713,E2 -25141.713} C_VEL
LIN {X 0,Y 126.434,Z 365.439,A -85,B 0,C 180,E1 -25145.708,E2 -25145.708} C_VEL
LIN {X 0,Y 126.553,Z 367.324,A -85,B 0,C 180,E1 -25148.969,E2 -25148.969} C_VEL
LIN {X 0,Y 127.401,Z 369.328,A -85,B 0,C 180,E1 -25154.18,E2 -25154.18} C_VEL
LIN {X 0,Y 129.291,Z 369.874,A -85,B 0,C 180,E1 -25159.553,E2 -25159.553} C_VEL
LIN {X 0,Y 131.658,Z 369.211,A -85,B 0,C 180,E1 -25164.042,E2 -25164.042} C_VEL
LIN {X 0,Y 134.973,Z 367.345,A -85,B 0,C 180,E1 -25168.62,E2 -25168.62} C_VEL
LIN {X 0,Y 138.89,Z 364.295,A -85,B 0,C 180,E1 -25172.908,E2 -25172.908} C_VEL
LIN {X 0,Y 143.493,Z 359.75,A -85,B 0,C 180,E1 -25176.931,E2 -25176.931} C_VEL
LIN {X 0,Y 147.726,Z 354.989,A -85,B 0,C 180,E1 -25179.952,E2 -25179.952} C_VEL
LIN {X 0,Y 151.313,Z 350.444,A -85,B 0,C 180,E1 -25182.205,E2 -25182.205} C_VEL
LIN {X 0,Y 154.671,Z 345.616,A -85,B 0,C 180,E1 -25184.179,E2 -25184.179} C_VEL
LIN {X 0,Y 156.519,Z 339.758,A -85,B 0,C 180,E1 -25187.026,E2 -25187.026} C_VEL
LIN {X 0,Y 157.615,Z 334.102,A -85,B 0,C 180,E1 -25189.725,E2 -25189.725} C_VEL
LIN {X 0,Y 157.702,Z 330.373,A -85,B 0,C 180,E1 -25191.672,E2 -25191.672} C_VEL
LIN {X 0,Y 156.385,Z 323.691,A -85,B 0,C 180,E1 -25196.134,E2 -25196.134} C_VEL
LIN {X 0,Y 154.639,Z 317.603,A -85,B 0,C 180,E1 -25200.998,E2 -25200.998} C_VEL
LIN {X 0,Y 154.085,Z 315.946,A -85,B 0,C 180,E1 -25202.614,E2 -25202.614} C_VEL
LIN {X 0,Y 153.037,Z 313.899,A -85,B 0,C 180,E1 -25205.27,E2 -25205.27} C_VEL
LIN {X 0,Y 151.52,Z 310.626,A -85,B 0,C 180,E1 -25210.692,E2 -25210.692} C_VEL
LIN {X 0,Y 150.942,Z 309.997,A -85,B 0,C 180,E1 -25213.462,E2 -25213.462} C_VEL
LIN {X 0,Y 150.599,Z 309.959,A -85,B 0,C 180,E1 -25219.066,E2 -25219.066} C_VEL
LIN {X 0,Y 151.485,Z 311.22,A -85,B 0,C 180,E1 -25224.68,E2 -25224.68} C_VEL
LIN {X 0,Y 152.355,Z 312.406,A -85,B 0,C 180,E1 -25227.47,E2 -25227.47} C_VEL
LIN {X 0,Y 155.375,Z 318.193,A -85,B 0,C 180,E1 -25234.43,E2 -25234.43} C_VEL
LIN {X 0,Y 157.623,Z 323.366,A -85,B 0,C 180,E1 -25238.625,E2 -25238.625} C_VEL
LIN {X 0,Y 158.876,Z 328.602,A -85,B 0,C 180,E1 -25241.57,E2 -25241.57} C_VEL
LIN {X 0,Y 158.499,Z 333.841,A -85,B 0,C 180,E1 -25243.601,E2 -25243.601} C_VEL
LIN {X 0,Y 157.419,Z 340.609,A -85,B 0,C 180,E1 -25246.058,E2 -25246.058} C_VEL
LIN {X 0,Y 156.7,Z 343.685,A -85,B 0,C 180,E1 -25247.124,E2 -25247.124} C_VEL
LIN {X 0,Y 152.659,Z 352.24,A -85,B 0,C 180,E1 -25249.871,E2 -25249.871} C_VEL
LIN {X 0,Y 150.241,Z 356.986,A -85,B 0,C 180,E1 -25251.698,E2 -25251.698} C_VEL
LIN {X 0,Y 145.53,Z 363.662,A -85,B 0,C 180,E1 -25254.584,E2 -25254.584} C_VEL
LIN {X 0,Y 141.967,Z 368.135,A -85,B 0,C 180,E1 -25257.007,E2 -25257.007} C_VEL
LIN {X 0,Y 138.835,Z 371.877,A -85,B 0,C 180,E1 -25259.588,E2 -25259.588} C_VEL
LIN {X 0,Y 134.795,Z 376.242,A -85,B 0,C 180,E1 -25263.694,E2 -25263.694} C_VEL
LIN {X 0,Y 131.458,Z 379.398,A -85,B 0,C 180,E1 -25268.023,E2 -25268.023} C_VEL
LIN {X 0,Y 129.644,Z 380.914,A -85,B 0,C 180,E1 -25271.019,E2 -25271.019} C_VEL
LIN {X 0,Y 128.357,Z 381.96,A -85,B 0,C 180,E1 -25274.112,E2 -25274.112} C_VEL
LIN {X 0,Y 127.441,Z 382.443,A -85,B 0,C 180,E1 -25277.257,E2 -25277.257} C_VEL
LIN {X 0,Y 126.892,Z 382.477,A -85,B 0,C 180,E1 -25280.436,E2 -25280.436} C_VEL
LIN {X 0,Y 126.796,Z 381.464,A -85,B 0,C 180,E1 -25286.108,E2 -25286.108} C_VEL
LIN {X 0,Y 127.115,Z 379.783,A -85,B 0,C 180,E1 -25290.001,E2 -25290.001} C_VEL
LIN {X 0,Y 127.222,Z 377.723,A -85,B 0,C 180,E1 -25293.167,E2 -25293.167} C_VEL
LIN {X 0,Y 127.794,Z 373.609,A -85,B 0,C 180,E1 -25297.903,E2 -25297.903} C_VEL
LIN {X 0,Y 129.796,Z 367.803,A -85,B 0,C 180,E1 -25302.67,E2 -25302.67} C_VEL
LIN {X 0,Y 131.213,Z 371.803,A -85,B 0,C 180,E1 -25308.746,E2 -25308.746} C_VEL
LIN {X 0,Y 134.546,Z 374.861,A -85,B 0,C 180,E1 -25314.701,E2 -25314.701} C_VEL
LIN {X 0,Y 139.647,Z 376.946,A -85,B 0,C 180,E1 -25320.217,E2 -25320.217} C_VEL
LIN {X 0,Y 146.209,Z 378.086,A -85,B 0,C 180,E1 -25325.228,E2 -25325.228} C_VEL
LIN {X 0,Y 154.19,Z 378.316,A -85,B 0,C 180,E1 -25329.653,E2 -25329.653} C_VEL
LIN {X 0,Y 163.538,Z 377.647,A -85,B 0,C 180,E1 -25333.441,E2 -25333.441} C_VEL
LIN {X 0,Y 173.776,Z 376.034,A -85,B 0,C 180,E1 -25336.718,E2 -25336.718} C_VEL
LIN {X 0,Y 174.906,Z 375.648,A -85,B 0,C 180,E1 -25337.809,E2 -25337.809} C_VEL
LIN {X 0,Y 164.794,Z 375.887,A -85,B 0,C 180,E1 -25341.074,E2 -25341.074} C_VEL
LIN {X 0,Y 156.711,Z 375.273,A -85,B 0,C 180,E1 -25344.338,E2 -25344.338} C_VEL
LIN {X 0,Y 148.367,Z 373.535,A -85,B 0,C 180,E1 -25348.597,E2 -25348.597} C_VEL
LIN {X 0,Y 146.013,Z 372.748,A -85,B 0,C 180,E1 -25350.041,E2 -25350.041} C_VEL
LIN {X 0,Y 142.524,Z 371.557,A -85,B 0,C 180,E1 -25351.873,E2 -25351.873} C_VEL
LIN {X 0,Y 135.782,Z 368.971,A -85,B 0,C 180,E1 -25354.672,E2 -25354.672} C_VEL
LIN {X 0,Y 129.677,Z 365.753,A -85,B 0,C 180,E1 -25357.739,E2 -25357.739} C_VEL
LIN {X 0,Y 127.289,Z 363.636,A -85,B 0,C 180,E1 -25359.961,E2 -25359.961} C_VEL
LIN {X 0,Y 123.717,Z 357.069,A -85,B 0,C 180,E1 -25366.866,E2 -25366.866} C_VEL
LIN {X 0,Y 121.994,Z 350.551,A -85,B 0,C 180,E1 -25372.553,E2 -25372.553} C_VEL
LIN {X 0,Y 121.43,Z 342.692,A -85,B 0,C 180,E1 -25378.342,E2 -25378.342} C_VEL
LIN {X 0,Y 121.44,Z 334.487,A -85,B 0,C 180,E1 -25383.318,E2 -25383.318} C_VEL
LIN {X 0,Y 121.752,Z 326.341,A -85,B 0,C 180,E1 -25387.463,E2 -25387.463} C_VEL
LIN {X 0,Y 122.575,Z 314.425,A -85,B 0,C 180,E1 -25392.448,E2 -25392.448} C_VEL
LIN {X 0,Y 123.616,Z 303.837,A -85,B 0,C 180,E1 -25396.049,E2 -25396.049} C_VEL
LIN {X 0,Y 124.589,Z 293.578,A -85,B 0,C 180,E1 -25398.927,E2 -25398.927} C_VEL
LIN {X 0,Y 121.972,Z 279.357,A -85,B 0,C 180,E1 -25401.925,E2 -25401.925} C_VEL
LIN {X 0,Y 121.015,Z 273.411,A -85,B 0,C 180,E1 -25403.043,E2 -25403.043} C_VEL
LIN {X 0,Y 121.176,Z 273.392,A -85,B 0,C 180,E1 -25411.466,E2 -25411.466} C_VEL
LIN {X 0,Y 121.588,Z 273.336,A -85,B 0,C 180,E1 -25415.978,E2 -25415.978} C_VEL
LIN {X 0,Y 121.793,Z 273.309,A -85,B 0,C 180,E1 -25421.395,E2 -25421.395} C_VEL
LIN {X 0,Y 121.836,Z 273.308,A -85,B 0,C 180,E1 -25426.194,E2 -25426.194} C_VEL
LIN {X 0,Y 121.854,Z 273.31,A -85,B 0,C 180,E1 -25430.621,E2 -25430.621} C_VEL
LIN {X 0,Y 121.909,Z 273.3,A -85,B 0,C 180,E1 -25434.795,E2 -25434.795} C_VEL
LIN {X 0,Y 121.928,Z 273.296,A -85,B 0,C 180,E1 -25439.839,E2 -25439.839} C_VEL
LIN {X 0,Y 121.983,Z 273.289,A -85,B 0,C 180,E1 -25446.215,E2 -25446.215} C_VEL
LIN {X 0,Y 122.048,Z 273.283,A -85,B 0,C 180,E1 -25449.787,E2 -25449.787} C_VEL
LIN {X 0,Y 122.242,Z 273.253,A -85,B 0,C 180,E1 -25456.704,E2 -25456.704} C_VEL
LIN {X 0,Y 122.335,Z 273.379,A -85,B 0,C 180,E1 -25457.818,E2 -25457.818} C_VEL
LIN {X 0,Y 123.175,Z 276.659,A -85,B 0,C 180,E1 -25461.799,E2 -25461.799} C_VEL
LIN {X 0,Y 124.591,Z 282.348,A -85,B 0,C 180,E1 -25468.383,E2 -25468.383} C_VEL
LIN {X 0,Y 124.322,Z 286.298,A -85,B 0,C 180,E1 -25472.429,E2 -25472.429} C_VEL
LIN {X 0,Y 124.279,Z 286.508,A -85,B 0,C 180,E1 -25472.633,E2 -25472.633} C_VEL
LIN {X 0,Y 126.322,Z 297.405,A -85,B 0,C 180,E1 -25474.388,E2 -25474.388} C_VEL
LIN {X 0,Y 127.698,Z 307.08,A -85,B 0,C 180,E1 -25476.319,E2 -25476.319} C_VEL
LIN {X 0,Y 128.548,Z 316.782,A -85,B 0,C 180,E1 -25478.647,E2 -25478.647} C_VEL
LIN {X 0,Y 128.705,Z 323.68,A -85,B 0,C 180,E1 -25480.609,E2 -25480.609} C_VEL
LIN {X 0,Y 126.475,Z 333.432,A -85,B 0,C 180,E1 -25483.66,E2 -25483.66} C_VEL
LIN {X 0,Y 124.709,Z 340.791,A -85,B 0,C 180,E1 -25486.654,E2 -25486.654} C_VEL
LIN {X 0,Y 123.004,Z 347.512,A -85,B 0,C 180,E1 -25490.048,E2 -25490.048} C_VEL
LIN {X 0,Y 121.933,Z 351.961,A -85,B 0,C 180,E1 -25492.746,E2 -25492.746} C_VEL
LIN {X 0,Y 120.635,Z 357.401,A -85,B 0,C 180,E1 -25496.84,E2 -25496.84} C_VEL
LIN {X 0,Y 119.884,Z 360.989,A -85,B 0,C 180,E1 -25500.179,E2 -25500.179} C_VEL
LIN {X 0,Y 119.38,Z 364.602,A -85,B 0,C 180,E1 -25504.492,E2 -25504.492} C_VEL
LIN {X 0,Y 119.582,Z 367.991,A -85,B 0,C 180,E1 -25510.277,E2 -25510.277} C_VEL
LIN {X 0,Y 120.679,Z 369.827,A -85,B 0,C 180,E1 -25515.665,E2 -25515.665} C_VEL
LIN {X 0,Y 122.691,Z 370.285,A -85,B 0,C 180,E1 -25520.941,E2 -25520.941} C_VEL
LIN {X 0,Y 126.081,Z 369.329,A -85,B 0,C 180,E1 -25526.733,E2 -25526.733} C_VEL
LIN {X 0,Y 129.201,Z 367.614,A -85,B 0,C 180,E1 -25530.688,E2 -25530.688} C_VEL
LIN {X 0,Y 133.492,Z 364.478,A -85,B 0,C 180,E1 -25535.09,E2 -25535.09} C_VEL
LIN {X 0,Y 138.585,Z 359.8,A -85,B 0,C 180,E1 -25539.207,E2 -25539.207} C_VEL
LIN {X 0,Y 142.78,Z 355.368,A -85,B 0,C 180,E1 -25542.031,E2 -25542.031} C_VEL
LIN {X 0,Y 147.311,Z 349.891,A -85,B 0,C 180,E1 -25544.691,E2 -25544.691} C_VEL
LIN {X 0,Y 149.282,Z 347.17,A -85,B 0,C 180,E1 -25545.892,E2 -25545.892} C_VEL
LIN {X 0,Y 151.577,Z 340.654,A -85,B 0,C 180,E1 -25549.311,E2 -25549.311} C_VEL
LIN {X 0,Y 152.647,Z 335.502,A -85,B 0,C 180,E1 -25552.06,E2 -25552.06} C_VEL
LIN {X 0,Y 152.099,Z 329.924,A -85,B 0,C 180,E1 -25556.025,E2 -25556.025} C_VEL
LIN {X 0,Y 150.945,Z 323.994,A -85,B 0,C 180,E1 -25561.022,E2 -25561.022} C_VEL
LIN {X 0,Y 150.16,Z 321.191,A -85,B 0,C 180,E1 -25564.025,E2 -25564.025} C_VEL
LIN {X 0,Y 148.64,Z 317.138,A -85,B 0,C 180,E1 -25570.902,E2 -25570.902} C_VEL
LIN {X 0,Y 148.174,Z 316.537,A -85,B 0,C 180,E1 -25573.718,E2 -25573.718} C_VEL
LIN {X 0,Y 147.938,Z 316.598,A -85,B 0,C 180,E1 -25579.423,E2 -25579.423} C_VEL
LIN {X 0,Y 148.881,Z 317.992,A -85,B 0,C 180,E1 -25585.141,E2 -25585.141} C_VEL
LIN {X 0,Y 149.625,Z 319.503,A -85,B 0,C 180,E1 -25588.015,E2 -25588.015} C_VEL
LIN {X 0,Y 151.708,Z 324.033,A -85,B 0,C 180,E1 -25593.773,E2 -25593.773} C_VEL
LIN {X 0,Y 153.565,Z 329.247,A -85,B 0,C 180,E1 -25598.16,E2 -25598.16} C_VEL
LIN {X 0,Y 154.13,Z 333.348,A -85,B 0,C 180,E1 -25600.632,E2 -25600.632} C_VEL
LIN {X 0,Y 152.818,Z 340.76,A -85,B 0,C 180,E1 -25603.617,E2 -25603.617} C_VEL
LIN {X 0,Y 151.634,Z 345.098,A -85,B 0,C 180,E1 -25605.292,E2 -25605.292} C_VEL
LIN {X 0,Y 148.25,Z 351.771,A -85,B 0,C 180,E1 -25607.504,E2 -25607.504} C_VEL
LIN {X 0,Y 144.789,Z 357.856,A -85,B 0,C 180,E1 -25609.973,E2 -25609.973} C_VEL
LIN {X 0,Y 139.838,Z 364.267,A -85,B 0,C 180,E1 -25612.908,E2 -25612.908} C_VEL
LIN {X 0,Y 136.088,Z 368.546,A -85,B 0,C 180,E1 -25615.384,E2 -25615.384} C_VEL
LIN {X 0,Y 132.754,Z 372.155,A -85,B 0,C 180,E1 -25618.035,E2 -25618.035} C_VEL
LIN {X 0,Y 128.448,Z 376.337,A -85,B 0,C 180,E1 -25622.285,E2 -25622.285} C_VEL
LIN {X 0,Y 124.888,Z 379.339,A -85,B 0,C 180,E1 -25626.802,E2 -25626.802} C_VEL
LIN {X 0,Y 122.931,Z 380.716,A -85,B 0,C 180,E1 -25629.939,E2 -25629.939} C_VEL
LIN {X 0,Y 121.496,Z 381.661,A -85,B 0,C 180,E1 -25633.189,E2 -25633.189} C_VEL
LIN {X 0,Y 120.495,Z 382.113,A -85,B 0,C 180,E1 -25636.509,E2 -25636.509} C_VEL
LIN {X 0,Y 119.885,Z 382.023,A -85,B 0,C 180,E1 -25639.871,E2 -25639.871} C_VEL
LIN {X 0,Y 119.747,Z 380.743,A -85,B 0,C 180,E1 -25646.143,E2 -25646.143} C_VEL
LIN {X 0,Y 120.049,Z 379.063,A -85,B 0,C 180,E1 -25650.001,E2 -25650.001} C_VEL
LIN {X 0,Y 120.177,Z 376.92,A -85,B 0,C 180,E1 -25653.353,E2 -25653.353} C_VEL
LIN {X 0,Y 120.814,Z 372.578,A -85,B 0,C 180,E1 -25658.363,E2 -25658.363} C_VEL
LIN {X 0,Y 122.423,Z 367.815,A -85,B 0,C 180,E1 -25662.432,E2 -25662.432} C_VEL
LIN {X 0,Y 123.347,Z 365.835,A -85,B 0,C 180,E1 -25663.931,E2 -25663.931} C_VEL
LIN {X 0,Y 124.802,Z 369.679,A -85,B 0,C 180,E1 -25669.748,E2 -25669.748} C_VEL
LIN {X 0,Y 128.337,Z 373.052,A -85,B 0,C 180,E1 -25675.983,E2 -25675.983} C_VEL
LIN {X 0,Y 133.681,Z 375.455,A -85,B 0,C 180,E1 -25681.718,E2 -25681.718} C_VEL
LIN {X 0,Y 140.541,Z 376.94,A -85,B 0,C 180,E1 -25686.876,E2 -25686.876} C_VEL
LIN {X 0,Y 148.822,Z 377.57,A -85,B 0,C 180,E1 -25691.388,E2 -25691.388} C_VEL
LIN {X 0,Y 158.481,Z 377.328,A -85,B 0,C 180,E1 -25695.198,E2 -25695.198} C_VEL
LIN {X 0,Y 163.65,Z 376.859,A -85,B 0,C 180,E1 -25696.893,E2 -25696.893} C_VEL
LIN {X 0,Y 164.222,Z 376.632,A -85,B 0,C 180,E1 -25697.839,E2 -25697.839} C_VEL
LIN {X 0,Y 155.716,Z 376.045,A -85,B 0,C 180,E1 -25700.812,E2 -25700.812} C_VEL
LIN {X 0,Y 146.545,Z 374.393,A -85,B 0,C 180,E1 -25704.866,E2 -25704.866} C_VEL
LIN {X 0,Y 138.511,Z 371.703,A -85,B 0,C 180,E1 -25709.51,E2 -25709.51} C_VEL
LIN {X 0,Y 131.915,Z 367.96,A -85,B 0,C 180,E1 -25714.773,E2 -25714.773} C_VEL
LIN {X 0,Y 127.289,Z 363.636,A -85,B 0,C 180,E1 -25719.961,E2 -25719.961} C_VEL
LIN {X 0,Y 125.208,Z 361.389,A -85,B 0,C 180,E1 -25722.245,E2 -25722.245} C_VEL
LIN {X 0,Y 120.675,Z 356.881,A -85,B 0,C 180,E1 -25725.766,E2 -25725.766} C_VEL
LIN {X 0,Y 116.592,Z 351.777,A -85,B 0,C 180,E1 -25729.414,E2 -25729.414} C_VEL
LIN {X 0,Y 115.316,Z 348.592,A -85,B 0,C 180,E1 -25731.842,E2 -25731.842} C_VEL
LIN {X 0,Y 114.701,Z 339.977,A -85,B 0,C 180,E1 -25738.245,E2 -25738.245} C_VEL
LIN {X 0,Y 114.69,Z 331.285,A -85,B 0,C 180,E1 -25743.514,E2 -25743.514} C_VEL
LIN {X 0,Y 115.042,Z 322.608,A -85,B 0,C 180,E1 -25747.901,E2 -25747.901} C_VEL
LIN {X 0,Y 115.85,Z 311.594,A -85,B 0,C 180,E1 -25752.542,E2 -25752.542} C_VEL
LIN {X 0,Y 116.892,Z 299.962,A -85,B 0,C 180,E1 -25756.505,E2 -25756.505} C_VEL
LIN {X 0,Y 117.449,Z 292.84,A -85,B 0,C 180,E1 -25758.536,E2 -25758.536} C_VEL
LIN {X 0,Y 114.882,Z 279.158,A -85,B 0,C 180,E1 -25761.535,E2 -25761.535} C_VEL
LIN {X 0,Y 114.072,Z 274.276,A -85,B 0,C 180,E1 -25762.457,E2 -25762.457} C_VEL
LIN {X 0,Y 114.077,Z 274.274,A -85,B 0,C 180,E1 -25770.4,E2 -25770.4} C_VEL
LIN {X 0,Y 114.569,Z 274.214,A -85,B 0,C 180,E1 -25777.11,E2 -25777.11} C_VEL
LIN {X 0,Y 114.727,Z 274.193,A -85,B 0,C 180,E1 -25782.683,E2 -25782.683} C_VEL
LIN {X 0,Y 114.787,Z 274.183,A -85,B 0,C 180,E1 -25787.662,E2 -25787.662} C_VEL
LIN {X 0,Y 114.785,Z 274.184,A -85,B 0,C 180,E1 -25792.747,E2 -25792.747} C_VEL
LIN {X 0,Y 114.856,Z 274.174,A -85,B 0,C 180,E1 -25798.944,E2 -25798.944} C_VEL
LIN {X 0,Y 114.948,Z 274.164,A -85,B 0,C 180,E1 -25806.509,E2 -25806.509} C_VEL
LIN {X 0,Y 115.059,Z 274.144,A -85,B 0,C 180,E1 -25814.045,E2 -25814.045} C_VEL
LIN {X 0,Y 115.136,Z 274.167,A -85,B 0,C 180,E1 -25815.867,E2 -25815.867} C_VEL
LIN {X 0,Y 116.296,Z 278.313,A -85,B 0,C 180,E1 -25821.31,E2 -25821.31} C_VEL
LIN {X 0,Y 117.688,Z 284.093,A -85,B 0,C 180,E1 -25828.288,E2 -25828.288} C_VEL
LIN {X 0,Y 117.534,Z 286.778,A -85,B 0,C 180,E1 -25831.178,E2 -25831.178} C_VEL
LIN {X 0,Y 119.788,Z 299.021,A -85,B 0,C 180,E1 -25833.363,E2 -25833.363} C_VEL
LIN {X 0,Y 121.093,Z 309.058,A -85,B 0,C 180,E1 -25835.526,E2 -25835.526} C_VEL
LIN {X 0,Y 121.838,Z 319.561,A -85,B 0,C 180,E1 -25838.312,E2 -25838.312} C_VEL
LIN {X 0,Y 121.911,Z 323.864,A -85,B 0,C 180,E1 -25839.655,E2 -25839.655} C_VEL
LIN {X 0,Y 119.381,Z 334.487,A -85,B 0,C 180,E1 -25843.194,E2 -25843.194} C_VEL
LIN {X 0,Y 117.377,Z 342.343,A -85,B 0,C 180,E1 -25846.661,E2 -25846.661} C_VEL
LIN {X 0,Y 116.019,Z 347.542,A -85,B 0,C 180,E1 -25849.461,E2 -25849.461} C_VEL
LIN {X 0,Y 114.615,Z 353.099,A -85,B 0,C 180,E1 -25853.105,E2 -25853.105} C_VEL
LIN {X 0,Y 113.326,Z 358.412,A -85,B 0,C 180,E1 -25857.478,E2 -25857.478} C_VEL
LIN {X 0,Y 112.51,Z 362.752,A -85,B 0,C 180,E1 -25862.07,E2 -25862.07} C_VEL
LIN {X 0,Y 112.265,Z 365.299,A -85,B 0,C 180,E1 -25865.528,E2 -25865.528} C_VEL
LIN {X 0,Y 112.349,Z 367.227,A -85,B 0,C 180,E1 -25868.722,E2 -25868.722} C_VEL
LIN {X 0,Y 112.907,Z 369.177,A -85,B 0,C 180,E1 -25873.212,E2 -25873.212} C_VEL
LIN {X 0,Y 114.138,Z 370.336,A -85,B 0,C 180,E1 -25877.637,E2 -25877.637} C_VEL
LIN {X 0,Y 116.362,Z 370.677,A -85,B 0,C 180,E1 -25882.844,E2 -25882.844} C_VEL
LIN {X 0,Y 119.601,Z 369.872,A -85,B 0,C 180,E1 -25888.071,E2 -25888.071} C_VEL
LIN {X 0,Y 123.638,Z 367.903,A -85,B 0,C 180,E1 -25892.951,E2 -25892.951} C_VEL
LIN {X 0,Y 128.929,Z 364.173,A -85,B 0,C 180,E1 -25897.923,E2 -25897.923} C_VEL
LIN {X 0,Y 133.946,Z 359.842,A -85,B 0,C 180,E1 -25901.65,E2 -25901.65} C_VEL
LIN {X 0,Y 138.538,Z 355.238,A -85,B 0,C 180,E1 -25904.549,E2 -25904.549} C_VEL
LIN {X 0,Y 142.894,Z 350.266,A -85,B 0,C 180,E1 -25906.939,E2 -25906.939} C_VEL
LIN {X 0,Y 143.893,Z 348.86,A -85,B 0,C 180,E1 -25907.643,E2 -25907.643} C_VEL
LIN {X 0,Y 146.366,Z 342.96,A -85,B 0,C 180,E1 -25911.022,E2 -25911.022} C_VEL
LIN {X 0,Y 147.346,Z 339.288,A -85,B 0,C 180,E1 -25913.151,E2 -25913.151} C_VEL
LIN {X 0,Y 147.206,Z 334.165,A -85,B 0,C 180,E1 -25917.263,E2 -25917.263} C_VEL
LIN {X 0,Y 146.797,Z 329.788,A -85,B 0,C 180,E1 -25921.371,E2 -25921.371} C_VEL
LIN {X 0,Y 146.34,Z 327.272,A -85,B 0,C 180,E1 -25924.131,E2 -25924.131} C_VEL
LIN {X 0,Y 145.322,Z 323.412,A -85,B 0,C 180,E1 -25931.154,E2 -25931.154} C_VEL
LIN {X 0,Y 144.914,Z 322.841,A -85,B 0,C 180,E1 -25934.08,E2 -25934.08} C_VEL
LIN {X 0,Y 144.787,Z 323.044,A -85,B 0,C 180,E1 -25939.863,E2 -25939.863} C_VEL
LIN {X 0,Y 145.785,Z 324.562,A -85,B 0,C 180,E1 -25945.713,E2 -25945.713} C_VEL
LIN {X 0,Y 147.214,Z 328.646,A -85,B 0,C 180,E1 -25951.678,E2 -25951.678} C_VEL
LIN {X 0,Y 147.827,Z 329.875,A -85,B 0,C 180,E1 -25953.318,E2 -25953.318} C_VEL
LIN {X 0,Y 149.177,Z 334.95,A -85,B 0,C 180,E1 -25957.767,E2 -25957.767} C_VEL
LIN {X 0,Y 149.29,Z 336.937,A -85,B 0,C 180,E1 -25959.104,E2 -25959.104} C_VEL
LIN {X 0,Y 148.553,Z 340.628,A -85,B 0,C 180,E1 -25960.804,E2 -25960.804} C_VEL
LIN {X 0,Y 146.691,Z 346.592,A -85,B 0,C 180,E1 -25963.347,E2 -25963.347} C_VEL
LIN {X 0,Y 144.171,Z 351.318,A -85,B 0,C 180,E1 -25965.022,E2 -25965.022} C_VEL
LIN {X 0,Y 139.459,Z 358.728,A -85,B 0,C 180,E1 -25968.108,E2 -25968.108} C_VEL
LIN {X 0,Y 135.28,Z 363.786,A -85,B 0,C 180,E1 -25970.476,E2 -25970.476} C_VEL
LIN {X 0,Y 130.325,Z 369.01,A -85,B 0,C 180,E1 -25973.617,E2 -25973.617} C_VEL
LIN {X 0,Y 126.772,Z 372.43,A -85,B 0,C 180,E1 -25976.332,E2 -25976.332} C_VEL
LIN {X 0,Y 122.193,Z 376.434,A -85,B 0,C 180,E1 -25980.733,E2 -25980.733} C_VEL
LIN {X 0,Y 118.384,Z 379.292,A -85,B 0,C 180,E1 -25985.446,E2 -25985.446} C_VEL
LIN {X 0,Y 116.272,Z 380.529,A -85,B 0,C 180,E1 -25988.736,E2 -25988.736} C_VEL
LIN {X 0,Y 114.674,Z 381.336,A -85,B 0,C 180,E1 -25992.156,E2 -25992.156} C_VEL
LIN {X 0,Y 113.58,Z 381.723,A -85,B 0,C 180,E1 -25995.67,E2 -25995.67} C_VEL
LIN {X 0,Y 112.874,Z 381.568,A -85,B 0,C 180,E1 -25999.235,E2 -25999.235} C_VEL
LIN {X 0,Y 112.597,Z 380.921,A -85,B 0,C 180,E1 -26002.829,E2 -26002.829} C_VEL
LIN {X 0,Y 112.736,Z 379.831,A -85,B 0,C 180,E1 -26006.426,E2 -26006.426} C_VEL
LIN {X 0,Y 112.992,Z 378.243,A -85,B 0,C 180,E1 -26010.001,E2 -26010.001} C_VEL
LIN {X 0,Y 113.135,Z 376.051,A -85,B 0,C 180,E1 -26013.562,E2 -26013.562} C_VEL
LIN {X 0,Y 113.828,Z 371.568,A -85,B 0,C 180,E1 -26018.776,E2 -26018.776} C_VEL
LIN {X 0,Y 116.081,Z 365.467,A -85,B 0,C 180,E1 -26024.016,E2 -26024.016} C_VEL
LIN {X 0,Y 116.997,Z 363.759,A -85,B 0,C 180,E1 -26025.347,E2 -26025.347} C_VEL
LIN {X 0,Y 118.503,Z 367.407,A -85,B 0,C 180,E1 -26030.846,E2 -26030.846} C_VEL
LIN {X 0,Y 122.238,Z 371.072,A -85,B 0,C 180,E1 -26037.385,E2 -26037.385} C_VEL
LIN {X 0,Y 127.862,Z 373.8,A -85,B 0,C 180,E1 -26043.344,E2 -26043.344} C_VEL
LIN {X 0,Y 135.449,Z 375.687,A -85,B 0,C 180,E1 -26048.895,E2 -26048.895} C_VEL
LIN {X 0,Y 143.629,Z 376.614,A -85,B 0,C 180,E1 -26053.24,E2 -26053.24} C_VEL
LIN {X 0,Y 153.589,Z 376.802,A -85,B 0,C 180,E1 -26057.067,E2 -26057.067} C_VEL
LIN {X 0,Y 150.286,Z 376.139,A -85,B 0,C 180,E1 -26059.103,E2 -26059.103} C_VEL
LIN {X 0,Y 140.804,Z 374.045,A -85,B 0,C 180,E1 -26063.205,E2 -26063.205} C_VEL
LIN {X 0,Y 132.492,Z 370.935,A -85,B 0,C 180,E1 -26067.965,E2 -26067.965} C_VEL
LIN {X 0,Y 125.623,Z 366.792,A -85,B 0,C 180,E1 -26073.413,E2 -26073.413} C_VEL
LIN {X 0,Y 120.862,Z 362.19,A -85,B 0,C 180,E1 -26078.768,E2 -26078.768} C_VEL
LIN {X 0,Y 117.065,Z 355.156,A -85,B 0,C 180,E1 -26086.106,E2 -26086.106} C_VEL
LIN {X 0,Y 115.316,Z 348.592,A -85,B 0,C 180,E1 -26091.842,E2 -26091.842} C_VEL
LIN {X 0,Y 114.238,Z 345.275,A -85,B 0,C 180,E1 -26094.226,E2 -26094.226} C_VEL
LIN {X 0,Y 111.216,Z 338.984,A -85,B 0,C 180,E1 -26097.817,E2 -26097.817} C_VEL
LIN {X 0,Y 108.515,Z 332.18,A -85,B 0,C 180,E1 -26101.374,E2 -26101.374} C_VEL
LIN {X 0,Y 108.024,Z 327.979,A -85,B 0,C 180,E1 -26103.624,E2 -26103.624} C_VEL
LIN {X 0,Y 108.422,Z 317.517,A -85,B 0,C 180,E1 -26108.856,E2 -26108.856} C_VEL
LIN {X 0,Y 109.379,Z 305.658,A -85,B 0,C 180,E1 -26113.695,E2 -26113.695} C_VEL
LIN {X 0,Y 110.496,Z 293.455,A -85,B 0,C 180,E1 -26117.68,E2 -26117.68} C_VEL
LIN {X 0,Y 108.065,Z 280.575,A -85,B 0,C 180,E1 -26120.71,E2 -26120.71} C_VEL
LIN {X 0,Y 107.128,Z 275.137,A -85,B 0,C 180,E1 -26121.909,E2 -26121.909} C_VEL
LIN {X 0,Y 107.092,Z 275.145,A -85,B 0,C 180,E1 -26131.669,E2 -26131.669} C_VEL
LIN {X 0,Y 107.533,Z 275.091,A -85,B 0,C 180,E1 -26138.345,E2 -26138.345} C_VEL
LIN {X 0,Y 107.657,Z 275.075,A -85,B 0,C 180,E1 -26145.898,E2 -26145.898} C_VEL
LIN {X 0,Y 107.685,Z 275.073,A -85,B 0,C 180,E1 -26151.553,E2 -26151.553} C_VEL
LIN {X 0,Y 107.792,Z 275.054,A -85,B 0,C 180,E1 -26158.56,E2 -26158.56} C_VEL
LIN {X 0,Y 107.913,Z 275.039,A -85,B 0,C 180,E1 -26166.997,E2 -26166.997} C_VEL
LIN {X 0,Y 108.029,Z 275.129,A -85,B 0,C 180,E1 -26173.948,E2 -26173.948} C_VEL
LIN {X 0,Y 109.399,Z 279.994,A -85,B 0,C 180,E1 -26180.757,E2 -26180.757} C_VEL
LIN {X 0,Y 110.795,Z 285.82,A -85,B 0,C 180,E1 -26188.182,E2 -26188.182} C_VEL
LIN {X 0,Y 110.764,Z 287.122,A -85,B 0,C 180,E1 -26189.659,E2 -26189.659} C_VEL
LIN {X 0,Y 112.851,Z 297.971,A -85,B 0,C 180,E1 -26191.682,E2 -26191.682} C_VEL
LIN {X 0,Y 113.926,Z 306.377,A -85,B 0,C 180,E1 -26193.536,E2 -26193.536} C_VEL
LIN {X 0,Y 114.75,Z 314.527,A -85,B 0,C 180,E1 -26195.682,E2 -26195.682} C_VEL
LIN {X 0,Y 115.091,Z 323.186,A -85,B 0,C 180,E1 -26198.338,E2 -26198.338} C_VEL
LIN {X 0,Y 114.594,Z 326.476,A -85,B 0,C 180,E1 -26199.35,E2 -26199.35} C_VEL
LIN {X 0,Y 112.303,Z 335.392,A -85,B 0,C 180,E1 -26202.652,E2 -26202.652} C_VEL
LIN {X 0,Y 110.324,Z 342.798,A -85,B 0,C 180,E1 -26206.137,E2 -26206.137} C_VEL
LIN {X 0,Y 108.601,Z 349.145,A -85,B 0,C 180,E1 -26209.861,E2 -26209.861} C_VEL
LIN {X 0,Y 107.042,Z 355.191,A -85,B 0,C 180,E1 -26214.309,E2 -26214.309} C_VEL
LIN {X 0,Y 105.653,Z 361.248,A -85,B 0,C 180,E1 -26220.144,E2 -26220.144} C_VEL
LIN {X 0,Y 105.214,Z 364.623,A -85,B 0,C 180,E1 -26224.458,E2 -26224.458} C_VEL
LIN {X 0,Y 105.289,Z 367.507,A -85,B 0,C 180,E1 -26229.354,E2 -26229.354} C_VEL
LIN {X 0,Y 105.738,Z 369.114,A -85,B 0,C 180,E1 -26233.018,E2 -26233.018} C_VEL
LIN {X 0,Y 107.464,Z 370.749,A -85,B 0,C 180,E1 -26239.156,E2 -26239.156} C_VEL
LIN {X 0,Y 110.585,Z 371.034,A -85,B 0,C 180,E1 -26245.709,E2 -26245.709} C_VEL
LIN {X 0,Y 113.821,Z 370.215,A -85,B 0,C 180,E1 -26250.398,E2 -26250.398} C_VEL
LIN {X 0,Y 118.273,Z 368.193,A -85,B 0,C 180,E1 -26255.42,E2 -26255.42} C_VEL
LIN {X 0,Y 123.506,Z 364.811,A -85,B 0,C 180,E1 -26260.036,E2 -26260.036} C_VEL
LIN {X 0,Y 129.588,Z 359.935,A -85,B 0,C 180,E1 -26264.266,E2 -26264.266} C_VEL
LIN {X 0,Y 134.885,Z 354.867,A -85,B 0,C 180,E1 -26267.373,E2 -26267.373} C_VEL
LIN {X 0,Y 138.067,Z 351.379,A -85,B 0,C 180,E1 -26269.048,E2 -26269.048} C_VEL
LIN {X 0,Y 140.193,Z 347.686,A -85,B 0,C 180,E1 -26271.35,E2 -26271.35} C_VEL
LIN {X 0,Y 141.535,Z 344.552,A -85,B 0,C 180,E1 -26273.269,E2 -26273.269} C_VEL
LIN {X 0,Y 142.049,Z 343.06,A -85,B 0,C 180,E1 -26274.321,E2 -26274.321} C_VEL
LIN {X 0,Y 142.263,Z 338.309,A -85,B 0,C 180,E1 -26278.584,E2 -26278.584} C_VEL
LIN {X 0,Y 142.179,Z 334.256,A -85,B 0,C 180,E1 -26282.833,E2 -26282.833} C_VEL
LIN {X 0,Y 141.99,Z 332.201,A -85,B 0,C 180,E1 -26285.681,E2 -26285.681} C_VEL
LIN {X 0,Y 141.544,Z 329.384,A -85,B 0,C 180,E1 -26291.455,E2 -26291.455} C_VEL
LIN {X 0,Y 141.255,Z 328.911,A -85,B 0,C 180,E1 -26294.404,E2 -26294.404} C_VEL
LIN {X 0,Y 141.228,Z 329.288,A -85,B 0,C 180,E1 -26300.386,E2 -26300.386} C_VEL
LIN {X 0,Y 141.612,Z 329.922,A -85,B 0,C 180,E1 -26303.392,E2 -26303.392} C_VEL
LIN {X 0,Y 142.247,Z 331.626,A -85,B 0,C 180,E1 -26307.212,E2 -26307.212} C_VEL
LIN {X 0,Y 143.533,Z 335.289,A -85,B 0,C 180,E1 -26312.589,E2 -26312.589} C_VEL
LIN {X 0,Y 144.32,Z 339.419,A -85,B 0,C 180,E1 -26316.697,E2 -26316.697} C_VEL
LIN {X 0,Y 144.361,Z 341.131,A -85,B 0,C 180,E1 -26317.94,E2 -26317.94} C_VEL
LIN {X 0,Y 142.392,Z 346.947,A -85,B 0,C 180,E1 -26320.747,E2 -26320.747} C_VEL
LIN {X 0,Y 141.404,Z 349.35,A -85,B 0,C 180,E1 -26321.796,E2 -26321.796} C_VEL
LIN {X 0,Y 136.259,Z 357.003,A -85,B 0,C 180,E1 -26324.83,E2 -26324.83} C_VEL
LIN {X 0,Y 132.149,Z 362.189,A -85,B 0,C 180,E1 -26327.307,E2 -26327.307} C_VEL
LIN {X 0,Y 126.729,Z 367.603,A -85,B 0,C 180,E1 -26330.376,E2 -26330.376} C_VEL
LIN {X 0,Y 120.914,Z 372.727,A -85,B 0,C 180,E1 -26334.462,E2 -26334.462} C_VEL
LIN {X 0,Y 116.045,Z 376.566,A -85,B 0,C 180,E1 -26339.017,E2 -26339.017} C_VEL
LIN {X 0,Y 111.956,Z 379.245,A -85,B 0,C 180,E1 -26343.933,E2 -26343.933} C_VEL
LIN {X 0,Y 109.675,Z 380.346,A -85,B 0,C 180,E1 -26347.389,E2 -26347.389} C_VEL
LIN {X 0,Y 107.899,Z 381.013,A -85,B 0,C 180,E1 -26350.994,E2 -26350.994} C_VEL
LIN {X 0,Y 106.699,Z 381.267,A -85,B 0,C 180,E1 -26354.724,E2 -26354.724} C_VEL
LIN {X 0,Y 105.892,Z 381.079,A -85,B 0,C 180,E1 -26358.516,E2 -26358.516} C_VEL
LIN {X 0,Y 105.55,Z 380.331,A -85,B 0,C 180,E1 -26362.348,E2 -26362.348} C_VEL
LIN {X 0,Y 105.654,Z 379.114,A -85,B 0,C 180,E1 -26366.186,E2 -26366.186} C_VEL
LIN {X 0,Y 105.937,Z 377.403,A -85,B 0,C 180,E1 -26370.001,E2 -26370.001} C_VEL
LIN {X 0,Y 106.097,Z 375.094,A -85,B 0,C 180,E1 -26373.799,E2 -26373.799} C_VEL
LIN {X 0,Y 106.48,Z 372.144,A -85,B 0,C 180,E1 -26377.586,E2 -26377.586} C_VEL
LIN {X 0,Y 107.94,Z 367.486,A -85,B 0,C 180,E1 -26382.217,E2 -26382.217} C_VEL
LIN {X 0,Y 109.955,Z 362.967,A -85,B 0,C 180,E1 -26385.795,E2 -26385.795} C_VEL
LIN {X 0,Y 110.812,Z 361.5,A -85,B 0,C 180,E1 -26386.855,E2 -26386.855} C_VEL
LIN {X 0,Y 113.108,Z 366.027,A -85,B 0,C 180,E1 -26393.822,E2 -26393.822} C_VEL
LIN {X 0,Y 119.026,Z 370.564,A -85,B 0,C 180,E1 -26402.102,E2 -26402.102} C_VEL
LIN {X 0,Y 125.763,Z 373.139,A -85,B 0,C 180,E1 -26407.932,E2 -26407.932} C_VEL
LIN {X 0,Y 134,Z 374.882,A -85,B 0,C 180,E1 -26412.987,E2 -26412.987} C_VEL
LIN {X 0,Y 143.649,Z 375.866,A -85,B 0,C 180,E1 -26417.213,E2 -26417.213} C_VEL
LIN {X 0,Y 139.965,Z 374.87,A -85,B 0,C 180,E1 -26419.25,E2 -26419.25} C_VEL
LIN {X 0,Y 130.31,Z 371.673,A -85,B 0,C 180,E1 -26423.999,E2 -26423.999} C_VEL
LIN {X 0,Y 122.848,Z 367.826,A -85,B 0,C 180,E1 -26429.011,E2 -26429.011} C_VEL
LIN {X 0,Y 116.375,Z 362.713,A -85,B 0,C 180,E1 -26434.993,E2 -26434.993} C_VEL
LIN {X 0,Y 112.015,Z 356.556,A -85,B 0,C 180,E1 -26441.718,E2 -26441.718} C_VEL
LIN {X 0,Y 109.304,Z 349.03,A -85,B 0,C 180,E1 -26448.879,E2 -26448.879} C_VEL
LIN {X 0,Y 108.128,Z 339.663,A -85,B 0,C 180,E1 -26456.274,E2 -26456.274} C_VEL
LIN {X 0,Y 108.003,Z 331.079,A -85,B 0,C 180,E1 -26461.865,E2 -26461.865} C_VEL
LIN {X 0,Y 108.024,Z 327.979,A -85,B 0,C 180,E1 -26463.624,E2 -26463.624} C_VEL
LIN {X 0,Y 107.591,Z 323.744,A -85,B 0,C 180,E1 -26465.739,E2 -26465.739} C_VEL
LIN {X 0,Y 106.323,Z 319.21,A -85,B 0,C 180,E1 -26467.64,E2 -26467.64} C_VEL
LIN {X 0,Y 103.305,Z 309.529,A -85,B 0,C 180,E1 -26471.172,E2 -26471.172} C_VEL
LIN {X 0,Y 102.613,Z 304.492,A -85,B 0,C 180,E1 -26472.986,E2 -26472.986} C_VEL
LIN {X 0,Y 102.645,Z 302.791,A -85,B 0,C 180,E1 -26473.613,E2 -26473.613} C_VEL
LIN {X 0,Y 103.487,Z 293.218,A -85,B 0,C 180,E1 -26476.878,E2 -26476.878} C_VEL
LIN {X 0,Y 100.931,Z 279.927,A -85,B 0,C 180,E1 -26480.145,E2 -26480.145} C_VEL
LIN {X 0,Y 100.225,Z 275.991,A -85,B 0,C 180,E1 -26481.1,E2 -26481.1} C_VEL
LIN {X 0,Y 100.073,Z 276.018,A -85,B 0,C 180,E1 -26492.567,E2 -26492.567} C_VEL
LIN {X 0,Y 100.478,Z 275.967,A -85,B 0,C 180,E1 -26499.698,E2 -26499.698} C_VEL
LIN {X 0,Y 100.625,Z 275.952,A -85,B 0,C 180,E1 -26505.697,E2 -26505.697} C_VEL
LIN {X 0,Y 100.623,Z 275.954,A -85,B 0,C 180,E1 -26511.052,E2 -26511.052} C_VEL
LIN {X 0,Y 100.689,Z 275.943,A -85,B 0,C 180,E1 -26516.888,E2 -26516.888} C_VEL
LIN {X 0,Y 100.788,Z 275.931,A -85,B 0,C 180,E1 -26525.267,E2 -26525.267} C_VEL
LIN {X 0,Y 100.92,Z 276.117,A -85,B 0,C 180,E1 -26531.736,E2 -26531.736} C_VEL
LIN {X 0,Y 102.13,Z 280.297,A -85,B 0,C 180,E1 -26538.085,E2 -26538.085} C_VEL
LIN {X 0,Y 103.143,Z 284.639,A -85,B 0,C 180,E1 -26544.133,E2 -26544.133} C_VEL
LIN {X 0,Y 103.884,Z 287.464,A -85,B 0,C 180,E1 -26547.877,E2 -26547.877} C_VEL
LIN {X 0,Y 105.818,Z 295.884,A -85,B 0,C 180,E1 -26549.571,E2 -26549.571} C_VEL
LIN {X 0,Y 107.141,Z 305.814,A -85,B 0,C 180,E1 -26551.86,E2 -26551.86} C_VEL
LIN {X 0,Y 107.936,Z 314.32,A -85,B 0,C 180,E1 -26554.208,E2 -26554.208} C_VEL
LIN {X 0,Y 108.272,Z 322.23,A -85,B 0,C 180,E1 -26556.76,E2 -26556.76} C_VEL
LIN {X 0,Y 108.172,Z 325.281,A -85,B 0,C 180,E1 -26557.81,E2 -26557.81} C_VEL
LIN {X 0,Y 105.559,Z 335.165,A -85,B 0,C 180,E1 -26561.521,E2 -26561.521} C_VEL
LIN {X 0,Y 103.725,Z 341.788,A -85,B 0,C 180,E1 -26564.719,E2 -26564.719} C_VEL
LIN {X 0,Y 101.972,Z 347.879,A -85,B 0,C 180,E1 -26568.333,E2 -26568.333} C_VEL
LIN {X 0,Y 100.374,Z 353.713,A -85,B 0,C 180,E1 -26572.649,E2 -26572.649} C_VEL
LIN {X 0,Y 99.034,Z 358.885,A -85,B 0,C 180,E1 -26577.469,E2 -26577.469} C_VEL
LIN {X 0,Y 98.416,Z 362.015,A -85,B 0,C 180,E1 -26581.025,E2 -26581.025} C_VEL
LIN {X 0,Y 98.091,Z 364.898,A -85,B 0,C 180,E1 -26584.972,E2 -26584.972} C_VEL
LIN {X 0,Y 98.252,Z 367.757,A -85,B 0,C 180,E1 -26590.073,E2 -26590.073} C_VEL
LIN {X 0,Y 99.051,Z 369.814,A -85,B 0,C 180,E1 -26595.196,E2 -26595.196} C_VEL
LIN {X 0,Y 101.033,Z 371.2,A -85,B 0,C 180,E1 -26601.239,E2 -26601.239} C_VEL
LIN {X 0,Y 102.845,Z 371.579,A -85,B 0,C 180,E1 -26605.087,E2 -26605.087} C_VEL
LIN {X 0,Y 105.771,Z 371.302,A -85,B 0,C 180,E1 -26609.745,E2 -26609.745} C_VEL
LIN {X 0,Y 109.307,Z 370.24,A -85,B 0,C 180,E1 -26614.177,E2 -26614.177} C_VEL
LIN {X 0,Y 113.425,Z 368.356,A -85,B 0,C 180,E1 -26618.344,E2 -26618.344} C_VEL
LIN {X 0,Y 118.947,Z 364.99,A -85,B 0,C 180,E1 -26622.816,E2 -26622.816} C_VEL
LIN {X 0,Y 125.493,Z 360.054,A -85,B 0,C 180,E1 -26627.055,E2 -26627.055} C_VEL
LIN {X 0,Y 132.619,Z 353.512,A -85,B 0,C 180,E1 -26630.852,E2 -26630.852} C_VEL
LIN {X 0,Y 134.61,Z 350.549,A -85,B 0,C 180,E1 -26632.743,E2 -26632.743} C_VEL
LIN {X 0,Y 136.263,Z 347.528,A -85,B 0,C 180,E1 -26634.821,E2 -26634.821} C_VEL
LIN {X 0,Y 136.596,Z 346.557,A -85,B 0,C 180,E1 -26635.573,E2 -26635.573} C_VEL
LIN {X 0,Y 137.255,Z 342.292,A -85,B 0,C 180,E1 -26640,E2 -26640} C_VEL
LIN {X 0,Y 137.445,Z 339.777,A -85,B 0,C 180,E1 -26642.931,E2 -26642.931} C_VEL
LIN {X 0,Y 137.563,Z 337.781,A -85,B 0,C 180,E1 -26645.864,E2 -26645.864} C_VEL
LIN {X 0,Y 137.394,Z 335.118,A -85,B 0,C 180,E1 -26651.806,E2 -26651.806} C_VEL
LIN {X 0,Y 137.206,Z 334.764,A -85,B 0,C 180,E1 -26654.839,E2 -26654.839} C_VEL
LIN {X 0,Y 137.291,Z 335.289,A -85,B 0,C 180,E1 -26660.998,E2 -26660.998} C_VEL
LIN {X 0,Y 137.637,Z 336.065,A -85,B 0,C 180,E1 -26664.11,E2 -26664.11} C_VEL
LIN {X 0,Y 138.045,Z 337.51,A -85,B 0,C 180,E1 -26667.271,E2 -26667.271} C_VEL
LIN {X 0,Y 138.948,Z 340.563,A -85,B 0,C 180,E1 -26672.079,E2 -26672.079} C_VEL
LIN {X 0,Y 139.268,Z 343.175,A -85,B 0,C 180,E1 -26675.01,E2 -26675.01} C_VEL
LIN {X 0,Y 139.127,Z 345.412,A -85,B 0,C 180,E1 -26676.897,E2 -26676.897} C_VEL
LIN {X 0,Y 136.759,Z 350.681,A -85,B 0,C 180,E1 -26679.57,E2 -26679.57} C_VEL
LIN {X 0,Y 131.379,Z 357.964,A -85,B 0,C 180,E1 -26682.647,E2 -26682.647} C_VEL
LIN {X 0,Y 128.179,Z 361.791,A -85,B 0,C 180,E1 -26684.538,E2 -26684.538} C_VEL
LIN {X 0,Y 123.631,Z 366.25,A -85,B 0,C 180,E1 -26686.988,E2 -26686.988} C_VEL
LIN {X 0,Y 119.222,Z 369.995,A -85,B 0,C 180,E1 -26689.577,E2 -26689.577} C_VEL
LIN {X 0,Y 113.721,Z 374.19,A -85,B 0,C 180,E1 -26693.679,E2 -26693.679} C_VEL
LIN {X 0,Y 108.424,Z 377.556,A -85,B 0,C 180,E1 -26698.765,E2 -26698.765} C_VEL
LIN {X 0,Y 105.602,Z 379.116,A -85,B 0,C 180,E1 -26702.234,E2 -26702.234} C_VEL
LIN {X 0,Y 103.151,Z 380.174,A -85,B 0,C 180,E1 -26705.871,E2 -26705.871} C_VEL
LIN {X 0,Y 101.177,Z 380.694,A -85,B 0,C 180,E1 -26709.678,E2 -26709.678} C_VEL
LIN {X 0,Y 99.839,Z 380.806,A -85,B 0,C 180,E1 -26713.646,E2 -26713.646} C_VEL
LIN {X 0,Y 98.942,Z 380.505,A -85,B 0,C 180,E1 -26717.697,E2 -26717.697} C_VEL
LIN {X 0,Y 98.529,Z 379.729,A -85,B 0,C 180,E1 -26721.799,E2 -26721.799} C_VEL
LIN {X 0,Y 98.609,Z 378.288,A -85,B 0,C 180,E1 -26726.196,E2 -26726.196} C_VEL
LIN {X 0,Y 98.938,Z 375.452,A -85,B 0,C 180,E1 -26732.036,E2 -26732.036} C_VEL
LIN {X 0,Y 99.518,Z 370.991,A -85,B 0,C 180,E1 -26738.12,E2 -26738.12} C_VEL
LIN {X 0,Y 101.126,Z 366.177,A -85,B 0,C 180,E1 -26743.055,E2 -26743.055} C_VEL
LIN {X 0,Y 103.539,Z 361.056,A -85,B 0,C 180,E1 -26747.152,E2 -26747.152} C_VEL
LIN {X 0,Y 104.746,Z 359.137,A -85,B 0,C 180,E1 -26748.575,E2 -26748.575} C_VEL
LIN {X 0,Y 108.084,Z 364.577,A -85,B 0,C 180,E1 -26757.076,E2 -26757.076} C_VEL
LIN {X 0,Y 113.353,Z 368.373,A -85,B 0,C 180,E1 -26763.919,E2 -26763.919} C_VEL
LIN {X 0,Y 120.434,Z 371.275,A -85,B 0,C 180,E1 -26769.935,E2 -26769.935} C_VEL
LIN {X 0,Y 129.03,Z 373.348,A -85,B 0,C 180,E1 -26775.08,E2 -26775.08} C_VEL
LIN {X 0,Y 133.805,Z 374.1,A -85,B 0,C 180,E1 -26777.337,E2 -26777.337} C_VEL
LIN {X 0,Y 129.771,Z 372.695,A -85,B 0,C 180,E1 -26779.467,E2 -26779.467} C_VEL
LIN {X 0,Y 118.84,Z 367.65,A -85,B 0,C 180,E1 -26785.819,E2 -26785.819} C_VEL
LIN {X 0,Y 111.709,Z 362.423,A -85,B 0,C 180,E1 -26791.846,E2 -26791.846} C_VEL
LIN {X 0,Y 106.597,Z 356.16,A -85,B 0,C 180,E1 -26798.739,E2 -26798.739} C_VEL
LIN {X 0,Y 103.332,Z 348.563,A -85,B 0,C 180,E1 -26806.229,E2 -26806.229} C_VEL
LIN {X 0,Y 101.676,Z 339.219,A -85,B 0,C 180,E1 -26814.049,E2 -26814.049} C_VEL
LIN {X 0,Y 101.371,Z 330.699,A -85,B 0,C 180,E1 -26820,E2 -26820} C_VEL
LIN {X 0,Y 101.504,Z 320.233,A -85,B 0,C 180,E1 -26825.962,E2 -26825.962} C_VEL
LIN {X 0,Y 102.196,Z 308.397,A -85,B 0,C 180,E1 -26831.404,E2 -26831.404} C_VEL
LIN {X 0,Y 102.645,Z 302.791,A -85,B 0,C 180,E1 -26833.613,E2 -26833.613} C_VEL
LIN {X 0,Y 102.135,Z 299.446,A -85,B 0,C 180,E1 -26834.708,E2 -26834.708} C_VEL
LIN {X 0,Y 99.994,Z 294.995,A -85,B 0,C 180,E1 -26835.829,E2 -26835.829} C_VEL
LIN {X 0,Y 96.054,Z 288.211,A -85,B 0,C 180,E1 -26837.292,E2 -26837.292} C_VEL
LIN {X 0,Y 94.843,Z 284.574,A -85,B 0,C 180,E1 -26838.147,E2 -26838.147} C_VEL
LIN {X 0,Y 93.386,Z 276.838,A -85,B 0,C 180,E1 -26840.08,E2 -26840.08} C_VEL
LIN {X 0,Y 93.08,Z 276.883,A -85,B 0,C 180,E1 -26853.843,E2 -26853.843} C_VEL
LIN {X 0,Y 93.411,Z 276.843,A -85,B 0,C 180,E1 -26861.202,E2 -26861.202} C_VEL
LIN {X 0,Y 93.528,Z 276.833,A -85,B 0,C 180,E1 -26868.716,E2 -26868.716} C_VEL
LIN {X 0,Y 93.586,Z 276.83,A -85,B 0,C 180,E1 -26875.698,E2 -26875.698} C_VEL
LIN {X 0,Y 93.67,Z 276.816,A -85,B 0,C 180,E1 -26884.206,E2 -26884.206} C_VEL
LIN {X 0,Y 93.763,Z 276.963,A -85,B 0,C 180,E1 -26888.855,E2 -26888.855} C_VEL
LIN {X 0,Y 94.782,Z 280.319,A -85,B 0,C 180,E1 -26894.569,E2 -26894.569} C_VEL
LIN {X 0,Y 95.989,Z 284.896,A -85,B 0,C 180,E1 -26901.579,E2 -26901.579} C_VEL
LIN {X 0,Y 96.642,Z 287.828,A -85,B 0,C 180,E1 -26905.698,E2 -26905.698} C_VEL
LIN {X 0,Y 98.586,Z 292.907,A -85,B 0,C 180,E1 -26907.072,E2 -26907.072} C_VEL
LIN {X 0,Y 100.219,Z 303.093,A -85,B 0,C 180,E1 -26909.447,E2 -26909.447} C_VEL
LIN {X 0,Y 101.187,Z 314.207,A -85,B 0,C 180,E1 -26912.627,E2 -26912.627} C_VEL
LIN {X 0,Y 101.482,Z 322.495,A -85,B 0,C 180,E1 -26915.464,E2 -26915.464} C_VEL
LIN {X 0,Y 101.495,Z 325.143,A -85,B 0,C 180,E1 -26916.46,E2 -26916.46} C_VEL
LIN {X 0,Y 98.628,Z 335.567,A -85,B 0,C 180,E1 -26920.586,E2 -26920.586} C_VEL
LIN {X 0,Y 96.891,Z 341.574,A -85,B 0,C 180,E1 -26923.635,E2 -26923.635} C_VEL
LIN {X 0,Y 94.647,Z 348.983,A -85,B 0,C 180,E1 -26928.395,E2 -26928.395} C_VEL
LIN {X 0,Y 92.99,Z 354.936,A -85,B 0,C 180,E1 -26933.268,E2 -26933.268} C_VEL
LIN {X 0,Y 91.725,Z 359.956,A -85,B 0,C 180,E1 -26938.473,E2 -26938.473} C_VEL
LIN {X 0,Y 91,Z 365.058,A -85,B 0,C 180,E1 -26945.396,E2 -26945.396} C_VEL
LIN {X 0,Y 91.091,Z 367.27,A -85,B 0,C 180,E1 -26949.507,E2 -26949.507} C_VEL
LIN {X 0,Y 92.266,Z 370.195,A -85,B 0,C 180,E1 -26956.721,E2 -26956.721} C_VEL
LIN {X 0,Y 95.106,Z 371.728,A -85,B 0,C 180,E1 -26964.376,E2 -26964.376} C_VEL
LIN {X 0,Y 98.316,Z 371.876,A -85,B 0,C 180,E1 -26969.974,E2 -26969.974} C_VEL
LIN {X 0,Y 102.922,Z 370.93,A -85,B 0,C 180,E1 -26975.813,E2 -26975.813} C_VEL
LIN {X 0,Y 108.37,Z 368.777,A -85,B 0,C 180,E1 -26981.079,E2 -26981.079} C_VEL
LIN {X 0,Y 114.721,Z 365.194,A -85,B 0,C 180,E1 -26985.815,E2 -26985.815} C_VEL
LIN {X 0,Y 119.92,Z 361.612,A -85,B 0,C 180,E1 -26989.005,E2 -26989.005} C_VEL
LIN {X 0,Y 125.921,Z 356.672,A -85,B 0,C 180,E1 -26992.165,E2 -26992.165} C_VEL
LIN {X 0,Y 127.482,Z 355.291,A -85,B 0,C 180,E1 -26992.899,E2 -26992.899} C_VEL
LIN {X 0,Y 129.336,Z 352.946,A -85,B 0,C 180,E1 -26994.543,E2 -26994.543} C_VEL
LIN {X 0,Y 131.152,Z 350.024,A -85,B 0,C 180,E1 -26996.928,E2 -26996.928} C_VEL
LIN {X 0,Y 132.093,Z 346.103,A -85,B 0,C 180,E1 -27001.524,E2 -27001.524} C_VEL
LIN {X 0,Y 132.681,Z 343.037,A -85,B 0,C 180,E1 -27006.081,E2 -27006.081} C_VEL
LIN {X 0,Y 132.904,Z 340.586,A -85,B 0,C 180,E1 -27012.211,E2 -27012.211} C_VEL
LIN {X 0,Y 132.785,Z 340.438,A -85,B 0,C 180,E1 -27017.694,E2 -27017.694} C_VEL
LIN {X 0,Y 132.989,Z 341.032,A -85,B 0,C 180,E1 -27021.711,E2 -27021.711} C_VEL
LIN {X 0,Y 133.378,Z 342.625,A -85,B 0,C 180,E1 -27026.393,E2 -27026.393} C_VEL
LIN {X 0,Y 134.027,Z 345.552,A -85,B 0,C 180,E1 -27031.626,E2 -27031.626} C_VEL
LIN {X 0,Y 134.097,Z 348.688,A -85,B 0,C 180,E1 -27035.205,E2 -27035.205} C_VEL
LIN {X 0,Y 132.293,Z 352.036,A -85,B 0,C 180,E1 -27037.168,E2 -27037.168} C_VEL
LIN {X 0,Y 130.203,Z 355.022,A -85,B 0,C 180,E1 -27038.494,E2 -27038.494} C_VEL
LIN {X 0,Y 124.508,Z 361.446,A -85,B 0,C 180,E1 -27041.59,E2 -27041.59} C_VEL
LIN {X 0,Y 118.565,Z 366.796,A -85,B 0,C 180,E1 -27044.659,E2 -27044.659} C_VEL
LIN {X 0,Y 111.769,Z 371.891,A -85,B 0,C 180,E1 -27048.683,E2 -27048.683} C_VEL
LIN {X 0,Y 108.971,Z 373.815,A -85,B 0,C 180,E1 -27050.708,E2 -27050.708} C_VEL
LIN {X 0,Y 105.884,Z 375.712,A -85,B 0,C 180,E1 -27053.319,E2 -27053.319} C_VEL
LIN {X 0,Y 102.409,Z 377.555,A -85,B 0,C 180,E1 -27056.701,E2 -27056.701} C_VEL
LIN {X 0,Y 99.341,Z 378.952,A -85,B 0,C 180,E1 -27060.316,E2 -27060.316} C_VEL
LIN {X 0,Y 96.686,Z 379.924,A -85,B 0,C 180,E1 -27064.143,E2 -27064.143} C_VEL
LIN {X 0,Y 94.52,Z 380.378,A -85,B 0,C 180,E1 -27068.176,E2 -27068.176} C_VEL
LIN {X 0,Y 93.004,Z 380.341,A -85,B 0,C 180,E1 -27072.407,E2 -27072.407} C_VEL
LIN {X 0,Y 91.995,Z 379.894,A -85,B 0,C 180,E1 -27076.752,E2 -27076.752} C_VEL
LIN {X 0,Y 91.514,Z 379.027,A -85,B 0,C 180,E1 -27081.165,E2 -27081.165} C_VEL
LIN {X 0,Y 91.574,Z 377.461,A -85,B 0,C 180,E1 -27086.112,E2 -27086.112} C_VEL
LIN {X 0,Y 91.834,Z 375.662,A -85,B 0,C 180,E1 -27090.001,E2 -27090.001} C_VEL
LIN {X 0,Y 92.179,Z 371.885,A -85,B 0,C 180,E1 -27096.15,E2 -27096.15} C_VEL
LIN {X 0,Y 93.482,Z 367.019,A -85,B 0,C 180,E1 -27101.932,E2 -27101.932} C_VEL
LIN {X 0,Y 95.968,Z 361.303,A -85,B 0,C 180,E1 -27107.034,E2 -27107.034} C_VEL
LIN {X 0,Y 98.83,Z 356.601,A -85,B 0,C 180,E1 -27110.49,E2 -27110.49} C_VEL
LIN {X 0,Y 102.276,Z 361.877,A -85,B 0,C 180,E1 -27118.752,E2 -27118.752} C_VEL
LIN {X 0,Y 107.881,Z 365.994,A -85,B 0,C 180,E1 -27125.897,E2 -27125.897} C_VEL
LIN {X 0,Y 115.312,Z 369.2,A -85,B 0,C 180,E1 -27132.101,E2 -27132.101} C_VEL
LIN {X 0,Y 124.273,Z 371.611,A -85,B 0,C 180,E1 -27137.324,E2 -27137.324} C_VEL
LIN {X 0,Y 113.368,Z 366.229,A -85,B 0,C 180,E1 -27143.699,E2 -27143.699} C_VEL
LIN {X 0,Y 105.727,Z 360.495,A -85,B 0,C 180,E1 -27150.096,E2 -27150.096} C_VEL
LIN {X 0,Y 100.348,Z 353.842,A -85,B 0,C 180,E1 -27157.344,E2 -27157.344} C_VEL
LIN {X 0,Y 96.9,Z 345.828,A -85,B 0,C 180,E1 -27165.295,E2 -27165.295} C_VEL
LIN {X 0,Y 95.204,Z 336.003,A -85,B 0,C 180,E1 -27173.643,E2 -27173.643} C_VEL
LIN {X 0,Y 94.832,Z 326.949,A -85,B 0,C 180,E1 -27180,E2 -27180} C_VEL
LIN {X 0,Y 94.901,Z 316.795,A -85,B 0,C 180,E1 -27185.845,E2 -27185.845} C_VEL
LIN {X 0,Y 95.629,Z 304.312,A -85,B 0,C 180,E1 -27191.661,E2 -27191.661} C_VEL
LIN {X 0,Y 96.476,Z 293.077,A -85,B 0,C 180,E1 -27195.854,E2 -27195.854} C_VEL
LIN {X 0,Y 95.217,Z 286.48,A -85,B 0,C 180,E1 -27197.67,E2 -27197.67} C_VEL
LIN {X 0,Y 94.843,Z 284.574,A -85,B 0,C 180,E1 -27198.147,E2 -27198.147} C_VEL
LIN {X 0,Y 93.89,Z 281.639,A -85,B 0,C 180,E1 -27199.389,E2 -27199.389} C_VEL
LIN {X 0,Y 92.521,Z 279.592,A -85,B 0,C 180,E1 -27201.139,E2 -27201.139} C_VEL
LIN {X 0,Y 91,Z 278.28,A -85,B 0,C 180,E1 -27203.238,E2 -27203.238} C_VEL
LIN {X 0,Y 88.815,Z 277.507,A -85,B 0,C 180,E1 -27206.834,E2 -27206.834} C_VEL
LIN {X 0,Y 86.298,Z 277.737,A -85,B 0,C 180,E1 -27213.799,E2 -27213.799} C_VEL
LIN {X 0,Y 86.056,Z 277.749,A -85,B 0,C 180,E1 -27216.702,E2 -27216.702} C_VEL
LIN {X 0,Y 86.377,Z 277.725,A -85,B 0,C 180,E1 -27222.921,E2 -27222.921} C_VEL
LIN {X 0,Y 86.452,Z 277.718,A -85,B 0,C 180,E1 -27229.431,E2 -27229.431} C_VEL
LIN {X 0,Y 86.529,Z 277.709,A -85,B 0,C 180,E1 -27235.35,E2 -27235.35} C_VEL
LIN {X 0,Y 86.622,Z 277.695,A -85,B 0,C 180,E1 -27245.017,E2 -27245.017} C_VEL
LIN {X 0,Y 87.53,Z 280.892,A -85,B 0,C 180,E1 -27251.265,E2 -27251.265} C_VEL
LIN {X 0,Y 88.757,Z 285.168,A -85,B 0,C 180,E1 -27258.582,E2 -27258.582} C_VEL
LIN {X 0,Y 89.456,Z 288.195,A -85,B 0,C 180,E1 -27263.224,E2 -27263.224} C_VEL
LIN {X 0,Y 92.566,Z 295.731,A -85,B 0,C 180,E1 -27265.56,E2 -27265.56} C_VEL
LIN {X 0,Y 93.986,Z 306.67,A -85,B 0,C 180,E1 -27268.506,E2 -27268.506} C_VEL
LIN {X 0,Y 94.6,Z 316.265,A -85,B 0,C 180,E1 -27271.587,E2 -27271.587} C_VEL
LIN {X 0,Y 94.743,Z 324.686,A -85,B 0,C 180,E1 -27274.786,E2 -27274.786} C_VEL
LIN {X 0,Y 94.174,Z 327.679,A -85,B 0,C 180,E1 -27275.889,E2 -27275.889} C_VEL
LIN {X 0,Y 91.512,Z 336.768,A -85,B 0,C 180,E1 -27279.95,E2 -27279.95} C_VEL
LIN {X 0,Y 89.449,Z 343.294,A -85,B 0,C 180,E1 -27283.633,E2 -27283.633} C_VEL
LIN {X 0,Y 87.205,Z 350.5,A -85,B 0,C 180,E1 -27288.806,E2 -27288.806} C_VEL
LIN {X 0,Y 85.292,Z 357.13,A -85,B 0,C 180,E1 -27294.986,E2 -27294.986} C_VEL
LIN {X 0,Y 84.157,Z 362.445,A -85,B 0,C 180,E1 -27301.605,E2 -27301.605} C_VEL
LIN {X 0,Y 83.957,Z 366.564,A -85,B 0,C 180,E1 -27308.572,E2 -27308.572} C_VEL
LIN {X 0,Y 84.668,Z 369.308,A -85,B 0,C 180,E1 -27314.874,E2 -27314.874} C_VEL
LIN {X 0,Y 85.692,Z 370.696,A -85,B 0,C 180,E1 -27318.995,E2 -27318.995} C_VEL
LIN {X 0,Y 88.639,Z 372.092,A -85,B 0,C 180,E1 -27326.287,E2 -27326.287} C_VEL
LIN {X 0,Y 90.164,Z 372.366,A -85,B 0,C 180,E1 -27329.026,E2 -27329.026} C_VEL
LIN {X 0,Y 93.68,Z 372.221,A -85,B 0,C 180,E1 -27334.191,E2 -27334.191} C_VEL
LIN {X 0,Y 97.889,Z 371.303,A -85,B 0,C 180,E1 -27338.962,E2 -27338.962} C_VEL
LIN {X 0,Y 103.887,Z 369.079,A -85,B 0,C 180,E1 -27344.299,E2 -27344.299} C_VEL
LIN {X 0,Y 108.062,Z 367.032,A -85,B 0,C 180,E1 -27347.303,E2 -27347.303} C_VEL
LIN {X 0,Y 113.899,Z 363.565,A -85,B 0,C 180,E1 -27350.845,E2 -27350.845} C_VEL
LIN {X 0,Y 120.131,Z 359.074,A -85,B 0,C 180,E1 -27354.013,E2 -27354.013} C_VEL
LIN {X 0,Y 123.021,Z 356.571,A -85,B 0,C 180,E1 -27355.441,E2 -27355.441} C_VEL
LIN {X 0,Y 124.493,Z 354.989,A -85,B 0,C 180,E1 -27356.763,E2 -27356.763} C_VEL
LIN {X 0,Y 125.607,Z 353.249,A -85,B 0,C 180,E1 -27358.396,E2 -27358.396} C_VEL
LIN {X 0,Y 126.953,Z 349.854,A -85,B 0,C 180,E1 -27363.173,E2 -27363.173} C_VEL
LIN {X 0,Y 127.555,Z 347.509,A -85,B 0,C 180,E1 -27367.36,E2 -27367.36} C_VEL
LIN {X 0,Y 128.088,Z 345.774,A -85,B 0,C 180,E1 -27372.678,E2 -27372.678} C_VEL
LIN {X 0,Y 128.036,Z 345.661,A -85,B 0,C 180,E1 -27375.929,E2 -27375.929} C_VEL
LIN {X 0,Y 128.196,Z 346.223,A -85,B 0,C 180,E1 -27381.255,E2 -27381.255} C_VEL
LIN {X 0,Y 128.488,Z 347.643,A -85,B 0,C 180,E1 -27385.949,E2 -27385.949} C_VEL
LIN {X 0,Y 128.819,Z 350.294,A -85,B 0,C 180,E1 -27391.218,E2 -27391.218} C_VEL
LIN {X 0,Y 128.749,Z 351.692,A -85,B 0,C 180,E1 -27393.084,E2 -27393.084} C_VEL
LIN {X 0,Y 128.053,Z 353.468,A -85,B 0,C 180,E1 -27394.588,E2 -27394.588} C_VEL
LIN {X 0,Y 125.951,Z 356.105,A -85,B 0,C 180,E1 -27395.993,E2 -27395.993} C_VEL
LIN {X 0,Y 119.932,Z 362.255,A -85,B 0,C 180,E1 -27399.064,E2 -27399.064} C_VEL
LIN {X 0,Y 113.719,Z 367.387,A -85,B 0,C 180,E1 -27402.131,E2 -27402.131} C_VEL
LIN {X 0,Y 108.837,Z 370.773,A -85,B 0,C 180,E1 -27404.74,E2 -27404.74} C_VEL
LIN {X 0,Y 102.997,Z 374.313,A -85,B 0,C 180,E1 -27408.641,E2 -27408.641} C_VEL
LIN {X 0,Y 100.272,Z 375.861,A -85,B 0,C 180,E1 -27410.891,E2 -27410.891} C_VEL
LIN {X 0,Y 96.545,Z 377.56,A -85,B 0,C 180,E1 -27414.384,E2 -27414.384} C_VEL
LIN {X 0,Y 93.21,Z 378.797,A -85,B 0,C 180,E1 -27418.144,E2 -27418.144} C_VEL
LIN {X 0,Y 90.325,Z 379.613,A -85,B 0,C 180,E1 -27422.171,E2 -27422.171} C_VEL
LIN {X 0,Y 87.94,Z 380.011,A -85,B 0,C 180,E1 -27426.448,E2 -27426.448} C_VEL
LIN {X 0,Y 86.228,Z 379.877,A -85,B 0,C 180,E1 -27430.973,E2 -27430.973} C_VEL
LIN {X 0,Y 85.087,Z 379.286,A -85,B 0,C 180,E1 -27435.654,E2 -27435.654} C_VEL
LIN {X 0,Y 84.509,Z 378.27,A -85,B 0,C 180,E1 -27440.426,E2 -27440.426} C_VEL
LIN {X 0,Y 84.54,Z 376.479,A -85,B 0,C 180,E1 -27446.017,E2 -27446.017} C_VEL
LIN {X 0,Y 84.786,Z 374.758,A -85,B 0,C 180,E1 -27450.001,E2 -27450.001} C_VEL
LIN {X 0,Y 85.144,Z 370.973,A -85,B 0,C 180,E1 -27456.355,E2 -27456.355} C_VEL
LIN {X 0,Y 86.661,Z 365.648,A -85,B 0,C 180,E1 -27462.887,E2 -27462.887} C_VEL
LIN {X 0,Y 89.358,Z 359.762,A -85,B 0,C 180,E1 -27468.337,E2 -27468.337} C_VEL
LIN {X 0,Y 92.772,Z 354.177,A -85,B 0,C 180,E1 -27472.259,E2 -27472.259} C_VEL
LIN {X 0,Y 93.116,Z 353.881,A -85,B 0,C 180,E1 -27472.547,E2 -27472.547} C_VEL
LIN {X 0,Y 97.949,Z 360.185,A -85,B 0,C 180,E1 -27482.558,E2 -27482.558} C_VEL
LIN {X 0,Y 106.296,Z 365.264,A -85,B 0,C 180,E1 -27491.39,E2 -27491.39} C_VEL
LIN {X 0,Y 114.901,Z 368.377,A -85,B 0,C 180,E1 -27497.223,E2 -27497.223} C_VEL
LIN {X 0,Y 105.61,Z 362.928,A -85,B 0,C 180,E1 -27503.208,E2 -27503.208} C_VEL
LIN {X 0,Y 98.254,Z 356.634,A -85,B 0,C 180,E1 -27509.954,E2 -27509.954} C_VEL
LIN {X 0,Y 92.664,Z 348.308,A -85,B 0,C 180,E1 -27518.884,E2 -27518.884} C_VEL
LIN {X 0,Y 89.913,Z 340.434,A -85,B 0,C 180,E1 -27526.439,E2 -27526.439} C_VEL
LIN {X 0,Y 88.789,Z 332.5,A -85,B 0,C 180,E1 -27533.182,E2 -27533.182} C_VEL
LIN {X 0,Y 88.363,Z 324.601,A -85,B 0,C 180,E1 -27538.861,E2 -27538.861} C_VEL
LIN {X 0,Y 88.345,Z 314.082,A -85,B 0,C 180,E1 -27545.135,E2 -27545.135} C_VEL
LIN {X 0,Y 88.899,Z 302.437,A -85,B 0,C 180,E1 -27550.823,E2 -27550.823} C_VEL
LIN {X 0,Y 89.584,Z 292.673,A -85,B 0,C 180,E1 -27554.705,E2 -27554.705} C_VEL
LIN {X 0,Y 86.985,Z 279.488,A -85,B 0,C 180,E1 -27558.314,E2 -27558.314} C_VEL
LIN {X 0,Y 86.618,Z 277.672,A -85,B 0,C 180,E1 -27558.803,E2 -27558.803} C_VEL
LIN {X 0,Y 85.695,Z 277.806,A -85,B 0,C 180,E1 -27569.478,E2 -27569.478} C_VEL
LIN {X 0,Y 86.068,Z 277.756,A -85,B 0,C 180,E1 -27575.256,E2 -27575.256} C_VEL
LIN {X 0,Y 86.056,Z 277.749,A -85,B 0,C 180,E1 -27576.702,E2 -27576.702} C_VEL
LIN {X 0,Y 85.45,Z 277.838,A -85,B 0,C 180,E1 -27580.616,E2 -27580.616} C_VEL
LIN {X 0,Y 83.969,Z 278.029,A -85,B 0,C 180,E1 -27584.509,E2 -27584.509} C_VEL
LIN {X 0,Y 79.665,Z 278.564,A -85,B 0,C 180,E1 -27595.479,E2 -27595.479} C_VEL
LIN {X 0,Y 79.373,Z 278.593,A -85,B 0,C 180,E1 -27598.406,E2 -27598.406} C_VEL
LIN {X 0,Y 79.482,Z 278.768,A -85,B 0,C 180,E1 -27601.203,E2 -27601.203} C_VEL
LIN {X 0,Y 80.273,Z 281.299,A -85,B 0,C 180,E1 -27606.796,E2 -27606.796} C_VEL
LIN {X 0,Y 81.094,Z 284.097,A -85,B 0,C 180,E1 -27612.427,E2 -27612.427} C_VEL
LIN {X 0,Y 82.305,Z 288.579,A -85,B 0,C 180,E1 -27620.272,E2 -27620.272} C_VEL
LIN {X 0,Y 86.491,Z 298.289,A -85,B 0,C 180,E1 -27623.892,E2 -27623.892} C_VEL
LIN {X 0,Y 87.549,Z 307.862,A -85,B 0,C 180,E1 -27626.764,E2 -27626.764} C_VEL
LIN {X 0,Y 87.999,Z 317.138,A -85,B 0,C 180,E1 -27629.999,E2 -27629.999} C_VEL
LIN {X 0,Y 88.027,Z 325.479,A -85,B 0,C 180,E1 -27633.432,E2 -27633.432} C_VEL
LIN {X 0,Y 85.846,Z 333.207,A -85,B 0,C 180,E1 -27636.751,E2 -27636.751} C_VEL
LIN {X 0,Y 82.666,Z 342.982,A -85,B 0,C 180,E1 -27642.271,E2 -27642.271} C_VEL
LIN {X 0,Y 80.424,Z 349.769,A -85,B 0,C 180,E1 -27647.393,E2 -27647.393} C_VEL
LIN {X 0,Y 78.564,Z 355.779,A -85,B 0,C 180,E1 -27653.194,E2 -27653.194} C_VEL
LIN {X 0,Y 77.239,Z 361.262,A -85,B 0,C 180,E1 -27660.029,E2 -27660.029} C_VEL
LIN {X 0,Y 76.816,Z 365.528,A -85,B 0,C 180,E1 -27666.98,E2 -27666.98} C_VEL
LIN {X 0,Y 77.289,Z 368.467,A -85,B 0,C 180,E1 -27673.326,E2 -27673.326} C_VEL
LIN {X 0,Y 79.629,Z 371.381,A -85,B 0,C 180,E1 -27682.591,E2 -27682.591} C_VEL
LIN {X 0,Y 82.756,Z 372.533,A -85,B 0,C 180,E1 -27689.366,E2 -27689.366} C_VEL
LIN {X 0,Y 87.426,Z 372.69,A -85,B 0,C 180,E1 -27696.3,E2 -27696.3} C_VEL
LIN {X 0,Y 93.18,Z 371.677,A -85,B 0,C 180,E1 -27702.44,E2 -27702.44} C_VEL
LIN {X 0,Y 100.48,Z 369.063,A -85,B 0,C 180,E1 -27708.297,E2 -27708.297} C_VEL
LIN {X 0,Y 107.278,Z 365.696,A -85,B 0,C 180,E1 -27712.471,E2 -27712.471} C_VEL
LIN {X 0,Y 112.823,Z 362.309,A -85,B 0,C 180,E1 -27715.327,E2 -27715.327} C_VEL
LIN {X 0,Y 117.729,Z 358.837,A -85,B 0,C 180,E1 -27717.519,E2 -27717.519} C_VEL
LIN {X 0,Y 118.972,Z 357.647,A -85,B 0,C 180,E1 -27718.476,E2 -27718.476} C_VEL
LIN {X 0,Y 120.036,Z 356.371,A -85,B 0,C 180,E1 -27720,E2 -27720} C_VEL
LIN {X 0,Y 121.187,Z 354.276,A -85,B 0,C 180,E1 -27723.324,E2 -27723.324} C_VEL
LIN {X 0,Y 121.992,Z 352.554,A -85,B 0,C 180,E1 -27726.616,E2 -27726.616} C_VEL
LIN {X 0,Y 122.507,Z 351.431,A -85,B 0,C 180,E1 -27729.91,E2 -27729.91} C_VEL
LIN {X 0,Y 122.88,Z 350.612,A -85,B 0,C 180,E1 -27733.518,E2 -27733.518} C_VEL
LIN {X 0,Y 122.849,Z 350.607,A -85,B 0,C 180,E1 -27736.621,E2 -27736.621} C_VEL
LIN {X 0,Y 122.945,Z 350.928,A -85,B 0,C 180,E1 -27740.058,E2 -27740.058} C_VEL
LIN {X 0,Y 123.07,Z 351.864,A -85,B 0,C 180,E1 -27743.98,E2 -27743.98} C_VEL
LIN {X 0,Y 123.188,Z 353.064,A -85,B 0,C 180,E1 -27747.155,E2 -27747.155} C_VEL
LIN {X 0,Y 123.276,Z 355.012,A -85,B 0,C 180,E1 -27751.223,E2 -27751.223} C_VEL
LIN {X 0,Y 122.948,Z 355.993,A -85,B 0,C 180,E1 -27752.483,E2 -27752.483} C_VEL
LIN {X 0,Y 121.944,Z 357.243,A -85,B 0,C 180,E1 -27753.314,E2 -27753.314} C_VEL
LIN {X 0,Y 114.347,Z 364.219,A -85,B 0,C 180,E1 -27756.965,E2 -27756.965} C_VEL
LIN {X 0,Y 106.5,Z 369.666,A -85,B 0,C 180,E1 -27760.634,E2 -27760.634} C_VEL
LIN {X 0,Y 99.21,Z 373.79,A -85,B 0,C 180,E1 -27764.896,E2 -27764.896} C_VEL
LIN {X 0,Y 94.848,Z 375.917,A -85,B 0,C 180,E1 -27768.174,E2 -27768.174} C_VEL
LIN {X 0,Y 90.861,Z 377.563,A -85,B 0,C 180,E1 -27771.773,E2 -27771.773} C_VEL
LIN {X 0,Y 87.232,Z 378.648,A -85,B 0,C 180,E1 -27775.67,E2 -27775.67} C_VEL
LIN {X 0,Y 84.091,Z 379.301,A -85,B 0,C 180,E1 -27779.904,E2 -27779.904} C_VEL
LIN {X 0,Y 81.458,Z 379.551,A -85,B 0,C 180,E1 -27784.445,E2 -27784.445} C_VEL
LIN {X 0,Y 79.524,Z 379.381,A -85,B 0,C 180,E1 -27789.299,E2 -27789.299} C_VEL
LIN {X 0,Y 78.223,Z 378.665,A -85,B 0,C 180,E1 -27794.364,E2 -27794.364} C_VEL
LIN {X 0,Y 77.533,Z 377.503,A -85,B 0,C 180,E1 -27799.556,E2 -27799.556} C_VEL
LIN {X 0,Y 77.508,Z 375.485,A -85,B 0,C 180,E1 -27805.876,E2 -27805.876} C_VEL
LIN {X 0,Y 77.759,Z 373.772,A -85,B 0,C 180,E1 -27810.001,E2 -27810.001} C_VEL
LIN {X 0,Y 78.117,Z 369.978,A -85,B 0,C 180,E1 -27816.592,E2 -27816.592} C_VEL
LIN {X 0,Y 79.42,Z 365.316,A -85,B 0,C 180,E1 -27822.782,E2 -27822.782} C_VEL
LIN {X 0,Y 81.757,Z 360.128,A -85,B 0,C 180,E1 -27828.126,E2 -27828.126} C_VEL
LIN {X 0,Y 85.436,Z 353.877,A -85,B 0,C 180,E1 -27833.001,E2 -27833.001} C_VEL
LIN {X 0,Y 87.608,Z 351.017,A -85,B 0,C 180,E1 -27834.861,E2 -27834.861} C_VEL
LIN {X 0,Y 92.601,Z 357.179,A -85,B 0,C 180,E1 -27844.697,E2 -27844.697} C_VEL
LIN {X 0,Y 101.463,Z 362.619,A -85,B 0,C 180,E1 -27853.843,E2 -27853.843} C_VEL
LIN {X 0,Y 105.78,Z 364.437,A -85,B 0,C 180,E1 -27856.958,E2 -27856.958} C_VEL
LIN {X 0,Y 97.526,Z 358.748,A -85,B 0,C 180,E1 -27863.034,E2 -27863.034} C_VEL
LIN {X 0,Y 91.006,Z 352.319,A -85,B 0,C 180,E1 -27869.87,E2 -27869.87} C_VEL
LIN {X 0,Y 86.111,Z 344.268,A -85,B 0,C 180,E1 -27878.453,E2 -27878.453} C_VEL
LIN {X 0,Y 83.377,Z 335.771,A -85,B 0,C 180,E1 -27886.597,E2 -27886.597} C_VEL
LIN {X 0,Y 82.325,Z 327.139,A -85,B 0,C 180,E1 -27893.875,E2 -27893.875} C_VEL
LIN {X 0,Y 81.854,Z 318.351,A -85,B 0,C 180,E1 -27900.001,E2 -27900.001} C_VEL
LIN {X 0,Y 81.886,Z 307.779,A -85,B 0,C 180,E1 -27906.159,E2 -27906.159} C_VEL
LIN {X 0,Y 82.51,Z 296.143,A -85,B 0,C 180,E1 -27911.672,E2 -27911.672} C_VEL
LIN {X 0,Y 82.721,Z 291.579,A -85,B 0,C 180,E1 -27913.512,E2 -27913.512} C_VEL
LIN {X 0,Y 79.89,Z 278.503,A -85,B 0,C 180,E1 -27917.402,E2 -27917.402} C_VEL
LIN {X 0,Y 78.759,Z 278.672,A -85,B 0,C 180,E1 -27932.372,E2 -27932.372} C_VEL
LIN {X 0,Y 79.086,Z 278.635,A -85,B 0,C 180,E1 -27938.468,E2 -27938.468} C_VEL
LIN {X 0,Y 79.327,Z 278.606,A -85,B 0,C 180,E1 -27945.135,E2 -27945.135} C_VEL
LIN {X 0,Y 79.384,Z 278.593,A -85,B 0,C 180,E1 -27952.825,E2 -27952.825} C_VEL
LIN {X 0,Y 79.373,Z 278.593,A -85,B 0,C 180,E1 -27958.406,E2 -27958.406} C_VEL
LIN {X 0,Y 78.995,Z 279.085,A -85,B 0,C 180,E1 -27960.728,E2 -27960.728} C_VEL
LIN {X 0,Y 77.655,Z 280.84,A -85,B 0,C 180,E1 -27963.748,E2 -27963.748} C_VEL
LIN {X 0,Y 74.704,Z 285.186,A -85,B 0,C 180,E1 -27969.767,E2 -27969.767} C_VEL
LIN {X 0,Y 74.494,Z 286.789,A -85,B 0,C 180,E1 -27972.631,E2 -27972.631} C_VEL
LIN {X 0,Y 75.029,Z 288.792,A -85,B 0,C 180,E1 -27976.628,E2 -27976.628} C_VEL
LIN {X 0,Y 78.977,Z 297.242,A -85,B 0,C 180,E1 -27980.389,E2 -27980.389} C_VEL
LIN {X 0,Y 80.568,Z 301.85,A -85,B 0,C 180,E1 -27982.323,E2 -27982.323} C_VEL
LIN {X 0,Y 81.305,Z 311.201,A -85,B 0,C 180,E1 -27985.499,E2 -27985.499} C_VEL
LIN {X 0,Y 81.485,Z 322.255,A -85,B 0,C 180,E1 -27989.999,E2 -27989.999} C_VEL
LIN {X 0,Y 81.352,Z 326.196,A -85,B 0,C 180,E1 -27991.856,E2 -27991.856} C_VEL
LIN {X 0,Y 78.497,Z 335.289,A -85,B 0,C 180,E1 -27996.108,E2 -27996.108} C_VEL
LIN {X 0,Y 75.931,Z 342.653,A -85,B 0,C 180,E1 -28000.667,E2 -28000.667} C_VEL
LIN {X 0,Y 73.332,Z 350.078,A -85,B 0,C 180,E1 -28006.708,E2 -28006.708} C_VEL
LIN {X 0,Y 71.809,Z 354.806,A -85,B 0,C 180,E1 -28011.531,E2 -28011.531} C_VEL
LIN {X 0,Y 70.409,Z 359.882,A -85,B 0,C 180,E1 -28018.044,E2 -28018.044} C_VEL
LIN {X 0,Y 69.851,Z 363.158,A -85,B 0,C 180,E1 -28023.14,E2 -28023.14} C_VEL
LIN {X 0,Y 69.892,Z 367.001,A -85,B 0,C 180,E1 -28030.813,E2 -28030.813} C_VEL
LIN {X 0,Y 70.522,Z 369.015,A -85,B 0,C 180,E1 -28035.765,E2 -28035.765} C_VEL
LIN {X 0,Y 73.086,Z 371.659,A -85,B 0,C 180,E1 -28044.762,E2 -28044.762} C_VEL
LIN {X 0,Y 78.012,Z 373.1,A -85,B 0,C 180,E1 -28054.273,E2 -28054.273} C_VEL
LIN {X 0,Y 82.502,Z 373.1,A -85,B 0,C 180,E1 -28060.077,E2 -28060.077} C_VEL
LIN {X 0,Y 88.856,Z 372.063,A -85,B 0,C 180,E1 -28066.273,E2 -28066.273} C_VEL
LIN {X 0,Y 96.086,Z 369.715,A -85,B 0,C 180,E1 -28071.588,E2 -28071.588} C_VEL
LIN {X 0,Y 104.213,Z 365.958,A -85,B 0,C 180,E1 -28076.133,E2 -28076.133} C_VEL
LIN {X 0,Y 112.903,Z 360.777,A -85,B 0,C 180,E1 -28080,E2 -28080} C_VEL
LIN {X 0,Y 114.449,Z 359.31,A -85,B 0,C 180,E1 -28081.759,E2 -28081.759} C_VEL
LIN {X 0,Y 115.132,Z 358.351,A -85,B 0,C 180,E1 -28083.499,E2 -28083.499} C_VEL
LIN {X 0,Y 116.257,Z 356.822,A -85,B 0,C 180,E1 -28086.944,E2 -28086.944} C_VEL
LIN {X 0,Y 116.947,Z 355.731,A -85,B 0,C 180,E1 -28090.386,E2 -28090.386} C_VEL
LIN {X 0,Y 117.375,Z 355.095,A -85,B 0,C 180,E1 -28093.857,E2 -28093.857} C_VEL
LIN {X 0,Y 117.364,Z 355.199,A -85,B 0,C 180,E1 -28097.422,E2 -28097.422} C_VEL
LIN {X 0,Y 117.444,Z 355.669,A -85,B 0,C 180,E1 -28101.041,E2 -28101.041} C_VEL
LIN {X 0,Y 117.509,Z 357.097,A -85,B 0,C 180,E1 -28106.219,E2 -28106.219} C_VEL
LIN {X 0,Y 117.534,Z 358.909,A -85,B 0,C 180,E1 -28110.461,E2 -28110.461} C_VEL
LIN {X 0,Y 114.186,Z 361.799,A -85,B 0,C 180,E1 -28112.19,E2 -28112.19} C_VEL
LIN {X 0,Y 110.25,Z 364.934,A -85,B 0,C 180,E1 -28114.035,E2 -28114.035} C_VEL
LIN {X 0,Y 104.769,Z 368.597,A -85,B 0,C 180,E1 -28116.393,E2 -28116.393} C_VEL
LIN {X 0,Y 96.827,Z 372.865,A -85,B 0,C 180,E1 -28120.349,E2 -28120.349} C_VEL
LIN {X 0,Y 89.667,Z 375.95,A -85,B 0,C 180,E1 -28125.138,E2 -28125.138} C_VEL
LIN {X 0,Y 85.392,Z 377.455,A -85,B 0,C 180,E1 -28128.821,E2 -28128.821} C_VEL
LIN {X 0,Y 81.444,Z 378.498,A -85,B 0,C 180,E1 -28132.84,E2 -28132.84} C_VEL
LIN {X 0,Y 78.013,Z 378.997,A -85,B 0,C 180,E1 -28137.281,E2 -28137.281} C_VEL
LIN {X 0,Y 75.094,Z 379.08,A -85,B 0,C 180,E1 -28142.1,E2 -28142.1} C_VEL
LIN {X 0,Y 72.908,Z 378.776,A -85,B 0,C 180,E1 -28147.321,E2 -28147.321} C_VEL
LIN {X 0,Y 71.413,Z 378.031,A -85,B 0,C 180,E1 -28152.829,E2 -28152.829} C_VEL
LIN {X 0,Y 70.588,Z 376.725,A -85,B 0,C 180,E1 -28158.515,E2 -28158.515} C_VEL
LIN {X 0,Y 70.487,Z 374.496,A -85,B 0,C 180,E1 -28165.605,E2 -28165.605} C_VEL
LIN {X 0,Y 70.753,Z 372.675,A -85,B 0,C 180,E1 -28170.001,E2 -28170.001} C_VEL
LIN {X 0,Y 71.296,Z 367.903,A -85,B 0,C 180,E1 -28178.504,E2 -28178.504} C_VEL
LIN {X 0,Y 73.117,Z 362.801,A -85,B 0,C 180,E1 -28185.328,E2 -28185.328} C_VEL
LIN {X 0,Y 76.348,Z 356.522,A -85,B 0,C 180,E1 -28191.606,E2 -28191.606} C_VEL
LIN {X 0,Y 80.259,Z 350.525,A -85,B 0,C 180,E1 -28195.967,E2 -28195.967} C_VEL
LIN {X 0,Y 82.325,Z 347.987,A -85,B 0,C 180,E1 -28197.465,E2 -28197.465} C_VEL
LIN {X 0,Y 87.468,Z 353.976,A -85,B 0,C 180,E1 -28207.056,E2 -28207.056} C_VEL
LIN {X 0,Y 96.89,Z 359.758,A -85,B 0,C 180,E1 -28216.5,E2 -28216.5} C_VEL
LIN {X 0,Y 95.149,Z 358.444,A -85,B 0,C 180,E1 -28218.336,E2 -28218.336} C_VEL
LIN {X 0,Y 87.066,Z 351.366,A -85,B 0,C 180,E1 -28225.595,E2 -28225.595} C_VEL
LIN {X 0,Y 80.734,Z 342.134,A -85,B 0,C 180,E1 -28235.576,E2 -28235.576} C_VEL
LIN {X 0,Y 77.58,Z 333.413,A -85,B 0,C 180,E1 -28244.231,E2 -28244.231} C_VEL
LIN {X 0,Y 76.21,Z 324.538,A -85,B 0,C 180,E1 -28252.049,E2 -28252.049} C_VEL
LIN {X 0,Y 75.555,Z 315.447,A -85,B 0,C 180,E1 -28258.668,E2 -28258.668} C_VEL
LIN {X 0,Y 75.437,Z 305.613,A -85,B 0,C 180,E1 -28264.677,E2 -28264.677} C_VEL
LIN {X 0,Y 75.889,Z 293.722,A -85,B 0,C 180,E1 -28270.675,E2 -28270.675} C_VEL
LIN {X 0,Y 75.9,Z 290.458,A -85,B 0,C 180,E1 -28272.026,E2 -28272.026} C_VEL
LIN {X 0,Y 73.287,Z 279.328,A -85,B 0,C 180,E1 -28275.504,E2 -28275.504} C_VEL
LIN {X 0,Y 71.563,Z 279.565,A -85,B 0,C 180,E1 -28289.41,E2 -28289.41} C_VEL
LIN {X 0,Y 72.031,Z 279.513,A -85,B 0,C 180,E1 -28298.687,E2 -28298.687} C_VEL
LIN {X 0,Y 72.211,Z 279.485,A -85,B 0,C 180,E1 -28307.055,E2 -28307.055} C_VEL
LIN {X 0,Y 72.293,Z 279.477,A -85,B 0,C 180,E1 -28314.316,E2 -28314.316} C_VEL
LIN {X 0,Y 72.621,Z 280.764,A -85,B 0,C 180,E1 -28318.508,E2 -28318.508} C_VEL
LIN {X 0,Y 73.46,Z 283.083,A -85,B 0,C 180,E1 -28324.498,E2 -28324.498} C_VEL
LIN {X 0,Y 74.494,Z 286.789,A -85,B 0,C 180,E1 -28332.631,E2 -28332.631} C_VEL
LIN {X 0,Y 75.076,Z 288.775,A -85,B 0,C 180,E1 -28335.132,E2 -28335.132} C_VEL
LIN {X 0,Y 75.812,Z 291.642,A -85,B 0,C 180,E1 -28337.07,E2 -28337.07} C_VEL
LIN {X 0,Y 76.64,Z 296.9,A -85,B 0,C 180,E1 -28339.16,E2 -28339.16} C_VEL
LIN {X 0,Y 76.44,Z 302.893,A -85,B 0,C 180,E1 -28340.7,E2 -28340.7} C_VEL
LIN {X 0,Y 75.072,Z 312.979,A -85,B 0,C 180,E1 -28343.51,E2 -28343.51} C_VEL
LIN {X 0,Y 74.979,Z 314.883,A -85,B 0,C 180,E1 -28344.288,E2 -28344.288} C_VEL
LIN {X 0,Y 74.877,Z 324.211,A -85,B 0,C 180,E1 -28348.655,E2 -28348.655} C_VEL
LIN {X 0,Y 74.722,Z 326.863,A -85,B 0,C 180,E1 -28349.999,E2 -28349.999} C_VEL
LIN {X 0,Y 71.422,Z 336.481,A -85,B 0,C 180,E1 -28354.938,E2 -28354.938} C_VEL
LIN {X 0,Y 68.467,Z 344.236,A -85,B 0,C 180,E1 -28360.38,E2 -28360.38} C_VEL
LIN {X 0,Y 66.01,Z 351.006,A -85,B 0,C 180,E1 -28366.619,E2 -28366.619} C_VEL
LIN {X 0,Y 64.307,Z 356.023,A -85,B 0,C 180,E1 -28372.488,E2 -28372.488} C_VEL
LIN {X 0,Y 63.352,Z 359.556,A -85,B 0,C 180,E1 -28377.44,E2 -28377.44} C_VEL
LIN {X 0,Y 62.692,Z 363.436,A -85,B 0,C 180,E1 -28384.09,E2 -28384.09} C_VEL
LIN {X 0,Y 62.907,Z 367.122,A -85,B 0,C 180,E1 -28392.091,E2 -28392.091} C_VEL
LIN {X 0,Y 64.221,Z 369.941,A -85,B 0,C 180,E1 -28399.999,E2 -28399.999} C_VEL
LIN {X 0,Y 67.105,Z 372.123,A -85,B 0,C 180,E1 -28408.421,E2 -28408.421} C_VEL
LIN {X 0,Y 71.845,Z 373.41,A -85,B 0,C 180,E1 -28416.965,E2 -28416.965} C_VEL
LIN {X 0,Y 74.547,Z 373.667,A -85,B 0,C 180,E1 -28420.518,E2 -28420.518} C_VEL
LIN {X 0,Y 79.673,Z 373.388,A -85,B 0,C 180,E1 -28426.004,E2 -28426.004} C_VEL
LIN {X 0,Y 85.435,Z 372.343,A -85,B 0,C 180,E1 -28430.797,E2 -28430.797} C_VEL
LIN {X 0,Y 92.917,Z 370.044,A -85,B 0,C 180,E1 -28435.662,E2 -28435.662} C_VEL
LIN {X 0,Y 98.425,Z 367.853,A -85,B 0,C 180,E1 -28438.515,E2 -28438.515} C_VEL
LIN {X 0,Y 105.462,Z 364.271,A -85,B 0,C 180,E1 -28441.621,E2 -28441.621} C_VEL
LIN {X 0,Y 108.031,Z 362.694,A -85,B 0,C 180,E1 -28442.656,E2 -28442.656} C_VEL
LIN {X 0,Y 108.832,Z 362.058,A -85,B 0,C 180,E1 -28443.702,E2 -28443.702} C_VEL
LIN {X 0,Y 110.236,Z 360.679,A -85,B 0,C 180,E1 -28447.325,E2 -28447.325} C_VEL
LIN {X 0,Y 111.117,Z 359.649,A -85,B 0,C 180,E1 -28450.938,E2 -28450.938} C_VEL
LIN {X 0,Y 111.582,Z 359.239,A -85,B 0,C 180,E1 -28454.592,E2 -28454.592} C_VEL
LIN {X 0,Y 111.586,Z 359.557,A -85,B 0,C 180,E1 -28459.137,E2 -28459.137} C_VEL
LIN {X 0,Y 111.597,Z 360.083,A -85,B 0,C 180,E1 -28462.201,E2 -28462.201} C_VEL
LIN {X 0,Y 111.594,Z 361.099,A -85,B 0,C 180,E1 -28466.158,E2 -28466.158} C_VEL
LIN {X 0,Y 111.547,Z 361.786,A -85,B 0,C 180,E1 -28468.108,E2 -28468.108} C_VEL
LIN {X 0,Y 110.601,Z 362.752,A -85,B 0,C 180,E1 -28469.106,E2 -28469.106} C_VEL
LIN {X 0,Y 103.578,Z 367.47,A -85,B 0,C 180,E1 -28471.989,E2 -28471.989} C_VEL
LIN {X 0,Y 95.089,Z 371.956,A -85,B 0,C 180,E1 -28475.61,E2 -28475.61} C_VEL
LIN {X 0,Y 89.753,Z 374.26,A -85,B 0,C 180,E1 -28478.461,E2 -28478.461} C_VEL
LIN {X 0,Y 84.763,Z 376.008,A -85,B 0,C 180,E1 -28481.737,E2 -28481.737} C_VEL
LIN {X 0,Y 80.165,Z 377.327,A -85,B 0,C 180,E1 -28485.465,E2 -28485.465} C_VEL
LIN {X 0,Y 75.889,Z 378.237,A -85,B 0,C 180,E1 -28489.59,E2 -28489.59} C_VEL
LIN {X 0,Y 72.128,Z 378.688,A -85,B 0,C 180,E1 -28494.224,E2 -28494.224} C_VEL
LIN {X 0,Y 68.88,Z 378.608,A -85,B 0,C 180,E1 -28499.326,E2 -28499.326} C_VEL
LIN {X 0,Y 64.671,Z 377.272,A -85,B 0,C 180,E1 -28510.974,E2 -28510.974} C_VEL
LIN {X 0,Y 63.657,Z 375.929,A -85,B 0,C 180,E1 -28517.244,E2 -28517.244} C_VEL
LIN {X 0,Y 63.468,Z 373.506,A -85,B 0,C 180,E1 -28525.271,E2 -28525.271} C_VEL
LIN {X 0,Y 63.742,Z 371.566,A -85,B 0,C 180,E1 -28530.001,E2 -28530.001} C_VEL
LIN {X 0,Y 63.993,Z 368.406,A -85,B 0,C 180,E1 -28536.306,E2 -28536.306} C_VEL
LIN {X 0,Y 65.431,Z 363.488,A -85,B 0,C 180,E1 -28543.986,E2 -28543.986} C_VEL
LIN {X 0,Y 68.17,Z 357.843,A -85,B 0,C 180,E1 -28550.662,E2 -28550.662} C_VEL
LIN {X 0,Y 71.967,Z 351.659,A -85,B 0,C 180,E1 -28556.07,E2 -28556.07} C_VEL
LIN {X 0,Y 75.572,Z 346.755,A -85,B 0,C 180,E1 -28559.226,E2 -28559.226} C_VEL
LIN {X 0,Y 77.345,Z 344.783,A -85,B 0,C 180,E1 -28560.362,E2 -28560.362} C_VEL
LIN {X 0,Y 84.35,Z 351.867,A -85,B 0,C 180,E1 -28571.803,E2 -28571.803} C_VEL
LIN {X 0,Y 88.242,Z 354.372,A -85,B 0,C 180,E1 -28575.793,E2 -28575.793} C_VEL
LIN {X 0,Y 87.421,Z 353.578,A -85,B 0,C 180,E1 -28577.665,E2 -28577.665} C_VEL
LIN {X 0,Y 79.237,Z 345.319,A -85,B 0,C 180,E1 -28586.335,E2 -28586.335} C_VEL
LIN {X 0,Y 73.876,Z 336.182,A -85,B 0,C 180,E1 -28596.153,E2 -28596.153} C_VEL
LIN {X 0,Y 71.035,Z 326.547,A -85,B 0,C 180,E1 -28605.68,E2 -28605.68} C_VEL
LIN {X 0,Y 69.854,Z 318.2,A -85,B 0,C 180,E1 -28612.776,E2 -28612.776} C_VEL
LIN {X 0,Y 69.195,Z 308.009,A -85,B 0,C 180,E1 -28620.001,E2 -28620.001} C_VEL
LIN {X 0,Y 69.245,Z 295.438,A -85,B 0,C 180,E1 -28627.289,E2 -28627.289} C_VEL
LIN {X 0,Y 69.314,Z 290.071,A -85,B 0,C 180,E1 -28629.853,E2 -28629.853} C_VEL
LIN {X 0,Y 66.89,Z 280.141,A -85,B 0,C 180,E1 -28633.042,E2 -28633.042} C_VEL
LIN {X 0,Y 64.54,Z 280.441,A -85,B 0,C 180,E1 -28645.823,E2 -28645.823} C_VEL
LIN {X 0,Y 64.57,Z 280.436,A -85,B 0,C 180,E1 -28652.972,E2 -28652.972} C_VEL
LIN {X 0,Y 64.996,Z 280.382,A -85,B 0,C 180,E1 -28660.806,E2 -28660.806} C_VEL
LIN {X 0,Y 65.151,Z 280.459,A -85,B 0,C 180,E1 -28666.73,E2 -28666.73} C_VEL
LIN {X 0,Y 65.824,Z 282.398,A -85,B 0,C 180,E1 -28674.037,E2 -28674.037} C_VEL
LIN {X 0,Y 66.634,Z 284.974,A -85,B 0,C 180,E1 -28681.774,E2 -28681.774} C_VEL
LIN {X 0,Y 67.495,Z 288.048,A -85,B 0,C 180,E1 -28689.578,E2 -28689.578} C_VEL
LIN {X 0,Y 67.93,Z 289.386,A -85,B 0,C 180,E1 -28692.244,E2 -28692.244} C_VEL
LIN {X 0,Y 72.269,Z 298.001,A -85,B 0,C 180,E1 -28697.06,E2 -28697.06} C_VEL
LIN {X 0,Y 74.421,Z 303.534,A -85,B 0,C 180,E1 -28699.89,E2 -28699.89} C_VEL
LIN {X 0,Y 75.014,Z 313.011,A -85,B 0,C 180,E1 -28703.51,E2 -28703.51} C_VEL
LIN {X 0,Y 74.979,Z 314.883,A -85,B 0,C 180,E1 -28704.288,E2 -28704.288} C_VEL
LIN {X 0,Y 74.574,Z 318.486,A -85,B 0,C 180,E1 -28705.726,E2 -28705.726} C_VEL
LIN {X 0,Y 72.847,Z 323.81,A -85,B 0,C 180,E1 -28707.594,E2 -28707.594} C_VEL
LIN {X 0,Y 70.249,Z 328.744,A -85,B 0,C 180,E1 -28709.396,E2 -28709.396} C_VEL
LIN {X 0,Y 64.487,Z 337.95,A -85,B 0,C 180,E1 -28713.873,E2 -28713.873} C_VEL
LIN {X 0,Y 63.028,Z 340.879,A -85,B 0,C 180,E1 -28715.888,E2 -28715.888} C_VEL
LIN {X 0,Y 59.64,Z 349.471,A -85,B 0,C 180,E1 -28723.631,E2 -28723.631} C_VEL
LIN {X 0,Y 57.278,Z 355.837,A -85,B 0,C 180,E1 -28731.597,E2 -28731.597} C_VEL
LIN {X 0,Y 55.891,Z 361.066,A -85,B 0,C 180,E1 -28740.196,E2 -28740.196} C_VEL
LIN {X 0,Y 55.63,Z 365.316,A -85,B 0,C 180,E1 -28749.172,E2 -28749.172} C_VEL
LIN {X 0,Y 56.597,Z 368.67,A -85,B 0,C 180,E1 -28758.162,E2 -28758.162} C_VEL
LIN {X 0,Y 58.878,Z 371.171,A -85,B 0,C 180,E1 -28766.672,E2 -28766.672} C_VEL
LIN {X 0,Y 62.316,Z 372.879,A -85,B 0,C 180,E1 -28774.452,E2 -28774.452} C_VEL
LIN {X 0,Y 67.001,Z 373.846,A -85,B 0,C 180,E1 -28781.658,E2 -28781.658} C_VEL
LIN {X 0,Y 73.873,Z 373.933,A -85,B 0,C 180,E1 -28789.031,E2 -28789.031} C_VEL
LIN {X 0,Y 81.644,Z 372.842,A -85,B 0,C 180,E1 -28795.061,E2 -28795.061} C_VEL
LIN {X 0,Y 91.368,Z 369.974,A -85,B 0,C 180,E1 -28800.557,E2 -28800.557} C_VEL
LIN {X 0,Y 99.49,Z 366.583,A -85,B 0,C 180,E1 -28804.05,E2 -28804.05} C_VEL
LIN {X 0,Y 103.153,Z 364.74,A -85,B 0,C 180,E1 -28805.865,E2 -28805.865} C_VEL
LIN {X 0,Y 103.934,Z 364.097,A -85,B 0,C 180,E1 -28807.772,E2 -28807.772} C_VEL
LIN {X 0,Y 105.061,Z 363.234,A -85,B 0,C 180,E1 -28811.577,E2 -28811.577} C_VEL
LIN {X 0,Y 105.519,Z 363.039,A -85,B 0,C 180,E1 -28815.451,E2 -28815.451} C_VEL
LIN {X 0,Y 105.517,Z 363.639,A -85,B 0,C 180,E1 -28821.177,E2 -28821.177} C_VEL
LIN {X 0,Y 105.445,Z 364.465,A -85,B 0,C 180,E1 -28825.175,E2 -28825.175} C_VEL
LIN {X 0,Y 105.224,Z 364.94,A -85,B 0,C 180,E1 -28826.603,E2 -28826.603} C_VEL
LIN {X 0,Y 100.02,Z 368.066,A -85,B 0,C 180,E1 -28828.559,E2 -28828.559} C_VEL
LIN {X 0,Y 91.152,Z 372.232,A -85,B 0,C 180,E1 -28831.993,E2 -28831.993} C_VEL
LIN {X 0,Y 85.521,Z 374.415,A -85,B 0,C 180,E1 -28834.737,E2 -28834.737} C_VEL
LIN {X 0,Y 80.21,Z 376.069,A -85,B 0,C 180,E1 -28837.948,E2 -28837.948} C_VEL
LIN {X 0,Y 75.253,Z 377.205,A -85,B 0,C 180,E1 -28841.659,E2 -28841.659} C_VEL
LIN {X 0,Y 70.619,Z 377.936,A -85,B 0,C 180,E1 -28845.843,E2 -28845.843} C_VEL
LIN {X 0,Y 66.488,Z 378.277,A -85,B 0,C 180,E1 -28850.639,E2 -28850.639} C_VEL
LIN {X 0,Y 62.861,Z 378.133,A -85,B 0,C 180,E1 -28856.014,E2 -28856.014} C_VEL
LIN {X 0,Y 58.017,Z 376.467,A -85,B 0,C 180,E1 -28868.691,E2 -28868.691} C_VEL
LIN {X 0,Y 56.8,Z 375.011,A -85,B 0,C 180,E1 -28875.673,E2 -28875.673} C_VEL
LIN {X 0,Y 56.467,Z 372.429,A -85,B 0,C 180,E1 -28884.673,E2 -28884.673} C_VEL
LIN {X 0,Y 56.727,Z 370.428,A -85,B 0,C 180,E1 -28890.001,E2 -28890.001} C_VEL
LIN {X 0,Y 57.686,Z 364.604,A -85,B 0,C 180,E1 -28901.596,E2 -28901.596} C_VEL
LIN {X 0,Y 60.471,Z 358.326,A -85,B 0,C 180,E1 -28910.407,E2 -28910.407} C_VEL
LIN {X 0,Y 63.821,Z 352.744,A -85,B 0,C 180,E1 -28916.136,E2 -28916.136} C_VEL
LIN {X 0,Y 67.085,Z 347.995,A -85,B 0,C 180,E1 -28919.844,E2 -28919.844} C_VEL
LIN {X 0,Y 72.085,Z 341.853,A -85,B 0,C 180,E1 -28923.26,E2 -28923.26} C_VEL
LIN {X 0,Y 72.672,Z 341.403,A -85,B 0,C 180,E1 -28923.578,E2 -28923.578} C_VEL
LIN {X 0,Y 79.896,Z 348.298,A -85,B 0,C 180,E1 -28934.727,E2 -28934.727} C_VEL
LIN {X 0,Y 81.014,Z 349.07,A -85,B 0,C 180,E1 -28936.052,E2 -28936.052} C_VEL
LIN {X 0,Y 72.444,Z 339.637,A -85,B 0,C 180,E1 -28946.095,E2 -28946.095} C_VEL
LIN {X 0,Y 67.704,Z 330.907,A -85,B 0,C 180,E1 -28955.468,E2 -28955.468} C_VEL
LIN {X 0,Y 65.157,Z 322.081,A -85,B 0,C 180,E1 -28964.357,E2 -28964.357} C_VEL
LIN {X 0,Y 63.964,Z 315.068,A -85,B 0,C 180,E1 -28970.514,E2 -28970.514} C_VEL
LIN {X 0,Y 63.103,Z 305.576,A -85,B 0,C 180,E1 -28977.607,E2 -28977.607} C_VEL
LIN {X 0,Y 62.894,Z 294.068,A -85,B 0,C 180,E1 -28984.808,E2 -28984.808} C_VEL
LIN {X 0,Y 62.829,Z 289.415,A -85,B 0,C 180,E1 -28987.23,E2 -28987.23} C_VEL
LIN {X 0,Y 60.572,Z 280.941,A -85,B 0,C 180,E1 -28990.235,E2 -28990.235} C_VEL
LIN {X 0,Y 58.588,Z 281.149,A -85,B 0,C 180,E1 -28996.326,E2 -28996.326} C_VEL
LIN {X 0,Y 57.525,Z 281.637,A -85,B 0,C 180,E1 -29009.256,E2 -29009.256} C_VEL
LIN {X 0,Y 57.903,Z 282.486,A -85,B 0,C 180,E1 -29017.365,E2 -29017.365} C_VEL
LIN {X 0,Y 58.849,Z 283.692,A -85,B 0,C 180,E1 -29025.771,E2 -29025.771} C_VEL
LIN {X 0,Y 59.605,Z 286.124,A -85,B 0,C 180,E1 -29035.627,E2 -29035.627} C_VEL
LIN {X 0,Y 60.45,Z 288.918,A -85,B 0,C 180,E1 -29044.522,E2 -29044.522} C_VEL
